//     PlcTask Inputs/GVL_iXlinker.EtherCAT_Master_EKxxxx.Beckhoff_EKM1xxx.Beckhoff_EKM1xxxEK1122.A_0004_EKM1101_0000_0019.MMS_Voltage_Us_In_Inputs.Status/Limit_2 <-> MMS Voltage Us In Inputs/Status/Limit 2
//     PlcTask Inputs/GVL_iXlinker.EtherCAT_Master_EKxxxx.Beckhoff_EKM1xxx.Beckhoff_EKM1xxxEK1122.A_0004_EKM1101_0000_0019.MMS_Voltage_Us_In_Inputs.Status/Error <-> MMS Voltage Us In Inputs/Status/Error
//     PlcTask Inputs/GVL_iXlinker.EtherCAT_Master_EKxxxx.Beckhoff_EKM1xxx.Beckhoff_EKM1xxxEK1122.A_0004_EKM1101_0000_0019.MMS_Voltage_Us_In_Inputs.Status/TxPDO_State <-> MMS Voltage Us In Inputs/Status/TxPDO State
//     PlcTask Inputs/GVL_iXlinker.EtherCAT_Master_EKxxxx.Beckhoff_EKM1xxx.Beckhoff_EKM1xxxEK1122.A_0004_EKM1101_0000_0019.MMS_Voltage_Us_In_Inputs.Status/TxPDO_Toggle <-> MMS Voltage Us In Inputs/Status/TxPDO Toggle
//     PlcTask Inputs/GVL_iXlinker.EtherCAT_Master_EKxxxx.Beckhoff_EKM1xxx.Beckhoff_EKM1xxxEK1122.A_0004_EKM1101_0000_0019.MMS_Voltage_Us_In_Inputs.Value <-> MMS Voltage Us In Inputs/Value
//     PlcTask Inputs/GVL_iXlinker.EtherCAT_Master_EKxxxx.Beckhoff_EKM1xxx.Beckhoff_EKM1xxxEK1122.A_0004_EKM1101_0000_0019.MMS_Voltage_Up_In_Inputs.Status/Underrange <-> MMS Voltage Up In Inputs/Status/Underrange
//     PlcTask Inputs/GVL_iXlinker.EtherCAT_Master_EKxxxx.Beckhoff_EKM1xxx.Beckhoff_EKM1xxxEK1122.A_0004_EKM1101_0000_0019.MMS_Voltage_Up_In_Inputs.Status/Overrange <-> MMS Voltage Up In Inputs/Status/Overrange
//     PlcTask Inputs/GVL_iXlinker.EtherCAT_Master_EKxxxx.Beckhoff_EKM1xxx.Beckhoff_EKM1xxxEK1122.A_0004_EKM1101_0000_0019.MMS_Voltage_Up_In_Inputs.Status/Limit_1 <-> MMS Voltage Up In Inputs/Status/Limit 1
//     PlcTask Inputs/GVL_iXlinker.EtherCAT_Master_EKxxxx.Beckhoff_EKM1xxx.Beckhoff_EKM1xxxEK1122.A_0004_EKM1101_0000_0019.MMS_Voltage_Up_In_Inputs.Status/Limit_2 <-> MMS Voltage Up In Inputs/Status/Limit 2
//     PlcTask Inputs/GVL_iXlinker.EtherCAT_Master_EKxxxx.Beckhoff_EKM1xxx.Beckhoff_EKM1xxxEK1122.A_0004_EKM1101_0000_0019.MMS_Voltage_Up_In_Inputs.Status/Error <-> MMS Voltage Up In Inputs/Status/Error
//     PlcTask Inputs/GVL_iXlinker.EtherCAT_Master_EKxxxx.Beckhoff_EKM1xxx.Beckhoff_EKM1xxxEK1122.A_0004_EKM1101_0000_0019.MMS_Voltage_Up_In_Inputs.Status/TxPDO_State <-> MMS Voltage Up In Inputs/Status/TxPDO State
//     PlcTask Inputs/GVL_iXlinker.EtherCAT_Master_EKxxxx.Beckhoff_EKM1xxx.Beckhoff_EKM1xxxEK1122.A_0004_EKM1101_0000_0019.MMS_Voltage_Up_In_Inputs.Status/TxPDO_Toggle <-> MMS Voltage Up In Inputs/Status/TxPDO Toggle
//     PlcTask Inputs/GVL_iXlinker.EtherCAT_Master_EKxxxx.Beckhoff_EKM1xxx.Beckhoff_EKM1xxxEK1122.A_0004_EKM1101_0000_0019.MMS_Voltage_Up_In_Inputs.Value <-> MMS Voltage Up In Inputs/Value
//     PlcTask Inputs/GVL_iXlinker.EtherCAT_Master_EKxxxx.Beckhoff_EKM1xxx.Beckhoff_EKM1xxxEK1122.A_0004_EKM1101_0000_0019.MMS_Voltage_Up_Out_Inputs.Status/Underrange <-> MMS Voltage Up Out Inputs/Status/Underrange
//     PlcTask Inputs/GVL_iXlinker.EtherCAT_Master_EKxxxx.Beckhoff_EKM1xxx.Beckhoff_EKM1xxxEK1122.A_0004_EKM1101_0000_0019.MMS_Voltage_Up_Out_Inputs.Status/Overrange <-> MMS Voltage Up Out Inputs/Status/Overrange
//     PlcTask Inputs/GVL_iXlinker.EtherCAT_Master_EKxxxx.Beckhoff_EKM1xxx.Beckhoff_EKM1xxxEK1122.A_0004_EKM1101_0000_0019.MMS_Voltage_Up_Out_Inputs.Status/Limit_1 <-> MMS Voltage Up Out Inputs/Status/Limit 1
//     PlcTask Inputs/GVL_iXlinker.EtherCAT_Master_EKxxxx.Beckhoff_EKM1xxx.Beckhoff_EKM1xxxEK1122.A_0004_EKM1101_0000_0019.MMS_Voltage_Up_Out_Inputs.Status/Limit_2 <-> MMS Voltage Up Out Inputs/Status/Limit 2
//     PlcTask Inputs/GVL_iXlinker.EtherCAT_Master_EKxxxx.Beckhoff_EKM1xxx.Beckhoff_EKM1xxxEK1122.A_0004_EKM1101_0000_0019.MMS_Voltage_Up_Out_Inputs.Status/Error <-> MMS Voltage Up Out Inputs/Status/Error
//     PlcTask Inputs/GVL_iXlinker.EtherCAT_Master_EKxxxx.Beckhoff_EKM1xxx.Beckhoff_EKM1xxxEK1122.A_0004_EKM1101_0000_0019.MMS_Voltage_Up_Out_Inputs.Status/TxPDO_State <-> MMS Voltage Up Out Inputs/Status/TxPDO State
//     PlcTask Inputs/GVL_iXlinker.EtherCAT_Master_EKxxxx.Beckhoff_EKM1xxx.Beckhoff_EKM1xxxEK1122.A_0004_EKM1101_0000_0019.MMS_Voltage_Up_Out_Inputs.Status/TxPDO_Toggle <-> MMS Voltage Up Out Inputs/Status/TxPDO Toggle
//     PlcTask Inputs/GVL_iXlinker.EtherCAT_Master_EKxxxx.Beckhoff_EKM1xxx.Beckhoff_EKM1xxxEK1122.A_0004_EKM1101_0000_0019.MMS_Voltage_Up_Out_Inputs.Value <-> MMS Voltage Up Out Inputs/Value
//     PlcTask Outputs/GVL_iXlinker.EtherCAT_Master_EKxxxx.Beckhoff_EKM1xxx.Beckhoff_EKM1xxxEK1122.A_0004_EKM1101_0000_0019.MMS_Device_Outputs.Control/Up_Out_OFF <-> MMS Device Outputs/Control/Up Out OFF
//     PlcTask Inputs/GVL_iXlinker.EtherCAT_Master_EKxxxx.Beckhoff_EKM1xxx.Beckhoff_EKM1xxxEK1122.A_0004_EKM1101_0000_0019.WcState.WcState <-> WcState/WcState
//     PlcTask Inputs/GVL_iXlinker.EtherCAT_Master_EKxxxx.Beckhoff_EKM1xxx.Beckhoff_EKM1xxxEK1122.A_0004_EKM1101_0000_0019.WcState.InputToggle <-> WcState/InputToggle
//     PlcTask Inputs/GVL_iXlinker.EtherCAT_Master_EKxxxx.Beckhoff_EKM1xxx.Beckhoff_EKM1xxxEK1122.A_0004_EKM1101_0000_0019.InfoData.AdsAddr <-> InfoData/AdsAddr
//     PlcTask Inputs/GVL_iXlinker.EtherCAT_Master_EKxxxx.Beckhoff_EKM1xxx.Beckhoff_EKM1xxxEK1122.A_0004_EKM1101_0000_0019.InfoData.DcOutputShift <-> InfoData/DcOutputShift
//     PlcTask Inputs/GVL_iXlinker.EtherCAT_Master_EKxxxx.Beckhoff_EKM1xxx.Beckhoff_EKM1xxxEK1122.A_0004_EKM1101_0000_0019.InfoData.DcInputShift <-> InfoData/DcInputShift
//     PlcTask Inputs/GVL_iXlinker.EtherCAT_Master_EKxxxx.Beckhoff_EKM1xxx.Beckhoff_EKM1xxxEK1122.A_0004_EKM1101_0000_0019.InfoData.State <-> InfoData/State
//   PLC/PLC Instance <-> EtherCAT Master EKxxxx/Beckhoff EKM1xxx/Beckhoff EKM1xxxEK1122/A_0005(EKM1101-0000-0020)
//     PlcTask Inputs/GVL_iXlinker.EtherCAT_Master_EKxxxx.Beckhoff_EKM1xxx.Beckhoff_EKM1xxxEK1122.A_0005_EKM1101_0000_0020.MMS_Device_Inputs.Status/Diag <-> MMS Device Inputs/Status/Diag
//     PlcTask Inputs/GVL_iXlinker.EtherCAT_Master_EKxxxx.Beckhoff_EKM1xxx.Beckhoff_EKM1xxxEK1122.A_0005_EKM1101_0000_0020.MMS_Device_Inputs.Status/Error <-> MMS Device Inputs/Status/Error
//     PlcTask Inputs/GVL_iXlinker.EtherCAT_Master_EKxxxx.Beckhoff_EKM1xxx.Beckhoff_EKM1xxxEK1122.A_0005_EKM1101_0000_0020.MMS_Device_Inputs.Status/Input_cycle_Counter <-> MMS Device Inputs/Status/Input cycle Counter
//     PlcTask Inputs/GVL_iXlinker.EtherCAT_Master_EKxxxx.Beckhoff_EKM1xxx.Beckhoff_EKM1xxxEK1122.A_0005_EKM1101_0000_0020.MMS_Device_Inputs.Status/TxPDO_State <-> MMS Device Inputs/Status/TxPDO State
//     PlcTask Inputs/GVL_iXlinker.EtherCAT_Master_EKxxxx.Beckhoff_EKM1xxx.Beckhoff_EKM1xxxEK1122.A_0005_EKM1101_0000_0020.MMS_Device_Inputs.Status/ID <-> MMS Device Inputs/Status/ID
//     PlcTask Inputs/GVL_iXlinker.EtherCAT_Master_EKxxxx.Beckhoff_EKM1xxx.Beckhoff_EKM1xxxEK1122.A_0005_EKM1101_0000_0020.MMS_Acceleration_Status.Status/Error <-> MMS Acceleration Status/Status/Error
//     PlcTask Inputs/GVL_iXlinker.EtherCAT_Master_EKxxxx.Beckhoff_EKM1xxx.Beckhoff_EKM1xxxEK1122.A_0005_EKM1101_0000_0020.MMS_Acceleration_Status.Status/Underrange <-> MMS Acceleration Status/Status/Underrange
//     PlcTask Inputs/GVL_iXlinker.EtherCAT_Master_EKxxxx.Beckhoff_EKM1xxx.Beckhoff_EKM1xxxEK1122.A_0005_EKM1101_0000_0020.MMS_Acceleration_Status.Status/Overrange <-> MMS Acceleration Status/Status/Overrange
//     PlcTask Inputs/GVL_iXlinker.EtherCAT_Master_EKxxxx.Beckhoff_EKM1xxx.Beckhoff_EKM1xxxEK1122.A_0005_EKM1101_0000_0020.MMS_Acceleration_Status.Status/Diag <-> MMS Acceleration Status/Status/Diag
//     PlcTask Inputs/GVL_iXlinker.EtherCAT_Master_EKxxxx.Beckhoff_EKM1xxx.Beckhoff_EKM1xxxEK1122.A_0005_EKM1101_0000_0020.MMS_Acceleration_Status.Status/Sensor_Ovr <-> MMS Acceleration Status/Status/Sensor Ovr
//     PlcTask Inputs/GVL_iXlinker.EtherCAT_Master_EKxxxx.Beckhoff_EKM1xxx.Beckhoff_EKM1xxxEK1122.A_0005_EKM1101_0000_0020.MMS_Acceleration_Status.Status/Overrun <-> MMS Acceleration Status/Status/Overrun
//     PlcTask Inputs/GVL_iXlinker.EtherCAT_Master_EKxxxx.Beckhoff_EKM1xxx.Beckhoff_EKM1xxxEK1122.A_0005_EKM1101_0000_0020.MMS_Acceleration_Status.Status/TxPDO_State <-> MMS Acceleration Status/Status/TxPDO State
//     PlcTask Inputs/GVL_iXlinker.EtherCAT_Master_EKxxxx.Beckhoff_EKM1xxx.Beckhoff_EKM1xxxEK1122.A_0005_EKM1101_0000_0020.MMS_Acceleration_Status.Number_of_samples <-> MMS Acceleration Status/Number of samples
//     PlcTask Inputs/GVL_iXlinker.EtherCAT_Master_EKxxxx.Beckhoff_EKM1xxx.Beckhoff_EKM1xxxEK1122.A_0005_EKM1101_0000_0020.MMS_Acceleration_X_Axis.Value <-> MMS Acceleration X-Axis/Value
//     PlcTask Inputs/GVL_iXlinker.EtherCAT_Master_EKxxxx.Beckhoff_EKM1xxx.Beckhoff_EKM1xxxEK1122.A_0005_EKM1101_0000_0020.MMS_Acceleration_Y_Axis.Value <-> MMS Acceleration Y-Axis/Value
//     PlcTask Inputs/GVL_iXlinker.EtherCAT_Master_EKxxxx.Beckhoff_EKM1xxx.Beckhoff_EKM1xxxEK1122.A_0005_EKM1101_0000_0020.MMS_Acceleration_Z_Axis.Value <-> MMS Acceleration Z-Axis/Value
//     PlcTask Inputs/GVL_iXlinker.EtherCAT_Master_EKxxxx.Beckhoff_EKM1xxx.Beckhoff_EKM1xxxEK1122.A_0005_EKM1101_0000_0020.MMS_Acceleration_Timestamp.Timestamp <-> MMS Acceleration Timestamp/Timestamp
//     PlcTask Inputs/GVL_iXlinker.EtherCAT_Master_EKxxxx.Beckhoff_EKM1xxx.Beckhoff_EKM1xxxEK1122.A_0005_EKM1101_0000_0020.MMS_Voltage_Us_In_Inputs.Status/Underrange <-> MMS Voltage Us In Inputs/Status/Underrange
//     PlcTask Inputs/GVL_iXlinker.EtherCAT_Master_EKxxxx.Beckhoff_EKM1xxx.Beckhoff_EKM1xxxEK1122.A_0005_EKM1101_0000_0020.MMS_Voltage_Us_In_Inputs.Status/Overrange <-> MMS Voltage Us In Inputs/Status/Overrange
//     PlcTask Inputs/GVL_iXlinker.EtherCAT_Master_EKxxxx.Beckhoff_EKM1xxx.Beckhoff_EKM1xxxEK1122.A_0005_EKM1101_0000_0020.MMS_Voltage_Us_In_Inputs.Status/Limit_1 <-> MMS Voltage Us In Inputs/Status/Limit 1
//     PlcTask Inputs/GVL_iXlinker.EtherCAT_Master_EKxxxx.Beckhoff_EKM1xxx.Beckhoff_EKM1xxxEK1122.A_0005_EKM1101_0000_0020.MMS_Voltage_Us_In_Inputs.Status/Limit_2 <-> MMS Voltage Us In Inputs/Status/Limit 2
//     PlcTask Inputs/GVL_iXlinker.EtherCAT_Master_EKxxxx.Beckhoff_EKM1xxx.Beckhoff_EKM1xxxEK1122.A_0005_EKM1101_0000_0020.MMS_Voltage_Us_In_Inputs.Status/Error <-> MMS Voltage Us In Inputs/Status/Error
//     PlcTask Inputs/GVL_iXlinker.EtherCAT_Master_EKxxxx.Beckhoff_EKM1xxx.Beckhoff_EKM1xxxEK1122.A_0005_EKM1101_0000_0020.MMS_Voltage_Us_In_Inputs.Status/TxPDO_State <-> MMS Voltage Us In Inputs/Status/TxPDO State
//     PlcTask Inputs/GVL_iXlinker.EtherCAT_Master_EKxxxx.Beckhoff_EKM1xxx.Beckhoff_EKM1xxxEK1122.A_0005_EKM1101_0000_0020.MMS_Voltage_Us_In_Inputs.Status/TxPDO_Toggle <-> MMS Voltage Us In Inputs/Status/TxPDO Toggle
//     PlcTask Inputs/GVL_iXlinker.EtherCAT_Master_EKxxxx.Beckhoff_EKM1xxx.Beckhoff_EKM1xxxEK1122.A_0005_EKM1101_0000_0020.MMS_Voltage_Us_In_Inputs.Value <-> MMS Voltage Us In Inputs/Value
//     PlcTask Inputs/GVL_iXlinker.EtherCAT_Master_EKxxxx.Beckhoff_EKM1xxx.Beckhoff_EKM1xxxEK1122.A_0005_EKM1101_0000_0020.MMS_Voltage_Up_In_Inputs.Status/Underrange <-> MMS Voltage Up In Inputs/Status/Underrange
//     PlcTask Inputs/GVL_iXlinker.EtherCAT_Master_EKxxxx.Beckhoff_EKM1xxx.Beckhoff_EKM1xxxEK1122.A_0005_EKM1101_0000_0020.MMS_Voltage_Up_In_Inputs.Status/Overrange <-> MMS Voltage Up In Inputs/Status/Overrange
//     PlcTask Inputs/GVL_iXlinker.EtherCAT_Master_EKxxxx.Beckhoff_EKM1xxx.Beckhoff_EKM1xxxEK1122.A_0005_EKM1101_0000_0020.MMS_Voltage_Up_In_Inputs.Status/Limit_1 <-> MMS Voltage Up In Inputs/Status/Limit 1
//     PlcTask Inputs/GVL_iXlinker.EtherCAT_Master_EKxxxx.Beckhoff_EKM1xxx.Beckhoff_EKM1xxxEK1122.A_0005_EKM1101_0000_0020.MMS_Voltage_Up_In_Inputs.Status/Limit_2 <-> MMS Voltage Up In Inputs/Status/Limit 2
//     PlcTask Inputs/GVL_iXlinker.EtherCAT_Master_EKxxxx.Beckhoff_EKM1xxx.Beckhoff_EKM1xxxEK1122.A_0005_EKM1101_0000_0020.MMS_Voltage_Up_In_Inputs.Status/Error <-> MMS Voltage Up In Inputs/Status/Error
//     PlcTask Inputs/GVL_iXlinker.EtherCAT_Master_EKxxxx.Beckhoff_EKM1xxx.Beckhoff_EKM1xxxEK1122.A_0005_EKM1101_0000_0020.MMS_Voltage_Up_In_Inputs.Status/TxPDO_State <-> MMS Voltage Up In Inputs/Status/TxPDO State
//     PlcTask Inputs/GVL_iXlinker.EtherCAT_Master_EKxxxx.Beckhoff_EKM1xxx.Beckhoff_EKM1xxxEK1122.A_0005_EKM1101_0000_0020.MMS_Voltage_Up_In_Inputs.Status/TxPDO_Toggle <-> MMS Voltage Up In Inputs/Status/TxPDO Toggle
//     PlcTask Inputs/GVL_iXlinker.EtherCAT_Master_EKxxxx.Beckhoff_EKM1xxx.Beckhoff_EKM1xxxEK1122.A_0005_EKM1101_0000_0020.MMS_Voltage_Up_In_Inputs.Value <-> MMS Voltage Up In Inputs/Value
//     PlcTask Inputs/GVL_iXlinker.EtherCAT_Master_EKxxxx.Beckhoff_EKM1xxx.Beckhoff_EKM1xxxEK1122.A_0005_EKM1101_0000_0020.MMS_Voltage_Up_Out_Inputs.Status/Underrange <-> MMS Voltage Up Out Inputs/Status/Underrange
//     PlcTask Inputs/GVL_iXlinker.EtherCAT_Master_EKxxxx.Beckhoff_EKM1xxx.Beckhoff_EKM1xxxEK1122.A_0005_EKM1101_0000_0020.MMS_Voltage_Up_Out_Inputs.Status/Overrange <-> MMS Voltage Up Out Inputs/Status/Overrange
//     PlcTask Inputs/GVL_iXlinker.EtherCAT_Master_EKxxxx.Beckhoff_EKM1xxx.Beckhoff_EKM1xxxEK1122.A_0005_EKM1101_0000_0020.MMS_Voltage_Up_Out_Inputs.Status/Limit_1 <-> MMS Voltage Up Out Inputs/Status/Limit 1
//     PlcTask Inputs/GVL_iXlinker.EtherCAT_Master_EKxxxx.Beckhoff_EKM1xxx.Beckhoff_EKM1xxxEK1122.A_0005_EKM1101_0000_0020.MMS_Voltage_Up_Out_Inputs.Status/Limit_2 <-> MMS Voltage Up Out Inputs/Status/Limit 2
//     PlcTask Inputs/GVL_iXlinker.EtherCAT_Master_EKxxxx.Beckhoff_EKM1xxx.Beckhoff_EKM1xxxEK1122.A_0005_EKM1101_0000_0020.MMS_Voltage_Up_Out_Inputs.Status/Error <-> MMS Voltage Up Out Inputs/Status/Error
//     PlcTask Inputs/GVL_iXlinker.EtherCAT_Master_EKxxxx.Beckhoff_EKM1xxx.Beckhoff_EKM1xxxEK1122.A_0005_EKM1101_0000_0020.MMS_Voltage_Up_Out_Inputs.Status/TxPDO_State <-> MMS Voltage Up Out Inputs/Status/TxPDO State
//     PlcTask Inputs/GVL_iXlinker.EtherCAT_Master_EKxxxx.Beckhoff_EKM1xxx.Beckhoff_EKM1xxxEK1122.A_0005_EKM1101_0000_0020.MMS_Voltage_Up_Out_Inputs.Status/TxPDO_Toggle <-> MMS Voltage Up Out Inputs/Status/TxPDO Toggle
//     PlcTask Inputs/GVL_iXlinker.EtherCAT_Master_EKxxxx.Beckhoff_EKM1xxx.Beckhoff_EKM1xxxEK1122.A_0005_EKM1101_0000_0020.MMS_Voltage_Up_Out_Inputs.Value <-> MMS Voltage Up Out Inputs/Value
//     PlcTask Outputs/GVL_iXlinker.EtherCAT_Master_EKxxxx.Beckhoff_EKM1xxx.Beckhoff_EKM1xxxEK1122.A_0005_EKM1101_0000_0020.MMS_Device_Outputs.Control/Up_Out_OFF <-> MMS Device Outputs/Control/Up Out OFF
//     PlcTask Inputs/GVL_iXlinker.EtherCAT_Master_EKxxxx.Beckhoff_EKM1xxx.Beckhoff_EKM1xxxEK1122.A_0005_EKM1101_0000_0020.WcState.WcState <-> WcState/WcState
//     PlcTask Inputs/GVL_iXlinker.EtherCAT_Master_EKxxxx.Beckhoff_EKM1xxx.Beckhoff_EKM1xxxEK1122.A_0005_EKM1101_0000_0020.WcState.InputToggle <-> WcState/InputToggle
//     PlcTask Inputs/GVL_iXlinker.EtherCAT_Master_EKxxxx.Beckhoff_EKM1xxx.Beckhoff_EKM1xxxEK1122.A_0005_EKM1101_0000_0020.InfoData.AdsAddr <-> InfoData/AdsAddr
//     PlcTask Inputs/GVL_iXlinker.EtherCAT_Master_EKxxxx.Beckhoff_EKM1xxx.Beckhoff_EKM1xxxEK1122.A_0005_EKM1101_0000_0020.InfoData.DcOutputShift <-> InfoData/DcOutputShift
//     PlcTask Inputs/GVL_iXlinker.EtherCAT_Master_EKxxxx.Beckhoff_EKM1xxx.Beckhoff_EKM1xxxEK1122.A_0005_EKM1101_0000_0020.InfoData.DcInputShift <-> InfoData/DcInputShift
//     PlcTask Inputs/GVL_iXlinker.EtherCAT_Master_EKxxxx.Beckhoff_EKM1xxx.Beckhoff_EKM1xxxEK1122.A_0005_EKM1101_0000_0020.InfoData.State <-> InfoData/State
//   PLC/PLC Instance <-> EtherCAT Master EKxxxx/Beckhoff EKx9xx
//     PlcTask Inputs/GVL_iXlinker.EtherCAT_Master_EKxxxx.Beckhoff_EKx9xx.InfoData.State <-> InfoData/State
//   PLC/PLC Instance <-> EtherCAT Master EKxxxx/Beckhoff EKx9xx/Beckhoff EKx9xxEK1122
//     PlcTask Inputs/GVL_iXlinker.EtherCAT_Master_EKxxxx.Beckhoff_EKx9xx.Beckhoff_EKx9xxEK1122.InfoData.State <-> InfoData/State
//   PLC/PLC Instance <-> EtherCAT Master EKxxxx/Beckhoff EKx9xx/Beckhoff EKx9xxEK1122/Beckhoff EKx9xxsub EK1100
//     PlcTask Inputs/GVL_iXlinker.EtherCAT_Master_EKxxxx.Beckhoff_EKx9xx.Beckhoff_EKx9xxEK1122.Beckhoff_EKx9xxsub_EK1100.InfoData.State <-> InfoData/State
//   PLC/PLC Instance <-> EtherCAT Master EKxxxx/Beckhoff EKx9xx/Beckhoff EKx9xxEK1122/A_0001(EK1960-0000-0019)
//     PlcTask Inputs/GVL_iXlinker.EtherCAT_Master_EKxxxx.Beckhoff_EKx9xx.Beckhoff_EKx9xxEK1122.A_0001_EK1960_0000_0019.Module_1_FSoE.FSoE_Inputs.FSOE/FSoE_Command <-> Module 1 (FSoE)/FSoE Inputs/FSOE/FSoE Command
//     PlcTask Inputs/GVL_iXlinker.EtherCAT_Master_EKxxxx.Beckhoff_EKx9xx.Beckhoff_EKx9xxEK1122.A_0001_EK1960_0000_0019.Module_1_FSoE.FSoE_Inputs.FSOE/FSOUT_Module_1_Module_Fault <-> Module 1 (FSoE)/FSoE Inputs/FSOE/FSOUT Module 1.Module Fault
//     PlcTask Inputs/GVL_iXlinker.EtherCAT_Master_EKxxxx.Beckhoff_EKx9xx.Beckhoff_EKx9xxEK1122.A_0001_EK1960_0000_0019.Module_1_FSoE.FSoE_Inputs.FSOE/FSOUT_Module_2_Module_Fault <-> Module 1 (FSoE)/FSoE Inputs/FSOE/FSOUT Module 2.Module Fault
//     PlcTask Inputs/GVL_iXlinker.EtherCAT_Master_EKxxxx.Beckhoff_EKx9xx.Beckhoff_EKx9xxEK1122.A_0001_EK1960_0000_0019.Module_1_FSoE.FSoE_Inputs.FSOE/FSOUT_Module_3_Module_Fault <-> Module 1 (FSoE)/FSoE Inputs/FSOE/FSOUT Module 3.Module Fault
//     PlcTask Inputs/GVL_iXlinker.EtherCAT_Master_EKxxxx.Beckhoff_EKx9xx.Beckhoff_EKx9xxEK1122.A_0001_EK1960_0000_0019.Module_1_FSoE.FSoE_Inputs.FSOE/FSOUT_Module_4_Module_Fault <-> Module 1 (FSoE)/FSoE Inputs/FSOE/FSOUT Module 4.Module Fault
//     PlcTask Inputs/GVL_iXlinker.EtherCAT_Master_EKxxxx.Beckhoff_EKx9xx.Beckhoff_EKx9xxEK1122.A_0001_EK1960_0000_0019.Module_1_FSoE.FSoE_Inputs.FSOE/FSOUT_Module_5_Module_Fault <-> Module 1 (FSoE)/FSoE Inputs/FSOE/FSOUT Module 5.Module Fault
//     PlcTask Inputs/GVL_iXlinker.EtherCAT_Master_EKxxxx.Beckhoff_EKx9xx.Beckhoff_EKx9xxEK1122.A_0001_EK1960_0000_0019.Module_1_FSoE.FSoE_Inputs.FSOE/FSOUT_Module_6_Module_Fault <-> Module 1 (FSoE)/FSoE Inputs/FSOE/FSOUT Module 6.Module Fault
//     PlcTask Inputs/GVL_iXlinker.EtherCAT_Master_EKxxxx.Beckhoff_EKx9xx.Beckhoff_EKx9xxEK1122.A_0001_EK1960_0000_0019.Module_1_FSoE.FSoE_Inputs.FSOE/FSIN_Module_1_Channel_1_Input <-> Module 1 (FSoE)/FSoE Inputs/FSOE/FSIN Module 1.Channel 1.Input
//     PlcTask Inputs/GVL_iXlinker.EtherCAT_Master_EKxxxx.Beckhoff_EKx9xx.Beckhoff_EKx9xxEK1122.A_0001_EK1960_0000_0019.Module_1_FSoE.FSoE_Inputs.FSOE/FSIN_Module_1_Channel_2_Input <-> Module 1 (FSoE)/FSoE Inputs/FSOE/FSIN Module 1.Channel 2.Input
//     PlcTask Inputs/GVL_iXlinker.EtherCAT_Master_EKxxxx.Beckhoff_EKx9xx.Beckhoff_EKx9xxEK1122.A_0001_EK1960_0000_0019.Module_1_FSoE.FSoE_Inputs.FSOE/FSIN_Module_2_Channel_1_Input <-> Module 1 (FSoE)/FSoE Inputs/FSOE/FSIN Module 2.Channel 1.Input
//     PlcTask Inputs/GVL_iXlinker.EtherCAT_Master_EKxxxx.Beckhoff_EKx9xx.Beckhoff_EKx9xxEK1122.A_0001_EK1960_0000_0019.Module_1_FSoE.FSoE_Inputs.FSOE/FSIN_Module_2_Channel_2_Input <-> Module 1 (FSoE)/FSoE Inputs/FSOE/FSIN Module 2.Channel 2.Input
//     PlcTask Inputs/GVL_iXlinker.EtherCAT_Master_EKxxxx.Beckhoff_EKx9xx.Beckhoff_EKx9xxEK1122.A_0001_EK1960_0000_0019.Module_1_FSoE.FSoE_Inputs.FSOE/FSIN_Module_3_Channel_1_Input <-> Module 1 (FSoE)/FSoE Inputs/FSOE/FSIN Module 3.Channel 1.Input
//     PlcTask Inputs/GVL_iXlinker.EtherCAT_Master_EKxxxx.Beckhoff_EKx9xx.Beckhoff_EKx9xxEK1122.A_0001_EK1960_0000_0019.Module_1_FSoE.FSoE_Inputs.FSOE/FSIN_Module_3_Channel_2_Input <-> Module 1 (FSoE)/FSoE Inputs/FSOE/FSIN Module 3.Channel 2.Input
//     PlcTask Inputs/GVL_iXlinker.EtherCAT_Master_EKxxxx.Beckhoff_EKx9xx.Beckhoff_EKx9xxEK1122.A_0001_EK1960_0000_0019.Module_1_FSoE.FSoE_Inputs.FSOE/FSIN_Module_4_Channel_1_Input <-> Module 1 (FSoE)/FSoE Inputs/FSOE/FSIN Module 4.Channel 1.Input
//     PlcTask Inputs/GVL_iXlinker.EtherCAT_Master_EKxxxx.Beckhoff_EKx9xx.Beckhoff_EKx9xxEK1122.A_0001_EK1960_0000_0019.Module_1_FSoE.FSoE_Inputs.FSOE/FSIN_Module_4_Channel_2_Input <-> Module 1 (FSoE)/FSoE Inputs/FSOE/FSIN Module 4.Channel 2.Input
//     PlcTask Inputs/GVL_iXlinker.EtherCAT_Master_EKxxxx.Beckhoff_EKx9xx.Beckhoff_EKx9xxEK1122.A_0001_EK1960_0000_0019.Module_1_FSoE.FSoE_Inputs.FSOE/FSIN_Module_5_Channel_1_Input <-> Module 1 (FSoE)/FSoE Inputs/FSOE/FSIN Module 5.Channel 1.Input
//     PlcTask Inputs/GVL_iXlinker.EtherCAT_Master_EKxxxx.Beckhoff_EKx9xx.Beckhoff_EKx9xxEK1122.A_0001_EK1960_0000_0019.Module_1_FSoE.FSoE_Inputs.FSOE/FSIN_Module_5_Channel_2_Input <-> Module 1 (FSoE)/FSoE Inputs/FSOE/FSIN Module 5.Channel 2.Input
//     PlcTask Inputs/GVL_iXlinker.EtherCAT_Master_EKxxxx.Beckhoff_EKx9xx.Beckhoff_EKx9xxEK1122.A_0001_EK1960_0000_0019.Module_1_FSoE.FSoE_Inputs.FSOE/FSIN_Module_6_Channel_1_Input <-> Module 1 (FSoE)/FSoE Inputs/FSOE/FSIN Module 6.Channel 1.Input
//     PlcTask Inputs/GVL_iXlinker.EtherCAT_Master_EKxxxx.Beckhoff_EKx9xx.Beckhoff_EKx9xxEK1122.A_0001_EK1960_0000_0019.Module_1_FSoE.FSoE_Inputs.FSOE/FSIN_Module_6_Channel_2_Input <-> Module 1 (FSoE)/FSoE Inputs/FSOE/FSIN Module 6.Channel 2.Input
//     PlcTask Inputs/GVL_iXlinker.EtherCAT_Master_EKxxxx.Beckhoff_EKx9xx.Beckhoff_EKx9xxEK1122.A_0001_EK1960_0000_0019.Module_1_FSoE.FSoE_Inputs.FSOE/FSIN_Module_7_Channel_1_Input <-> Module 1 (FSoE)/FSoE Inputs/FSOE/FSIN Module 7.Channel 1.Input
//     PlcTask Inputs/GVL_iXlinker.EtherCAT_Master_EKxxxx.Beckhoff_EKx9xx.Beckhoff_EKx9xxEK1122.A_0001_EK1960_0000_0019.Module_1_FSoE.FSoE_Inputs.FSOE/FSIN_Module_7_Channel_2_Input <-> Module 1 (FSoE)/FSoE Inputs/FSOE/FSIN Module 7.Channel 2.Input
//     PlcTask Inputs/GVL_iXlinker.EtherCAT_Master_EKxxxx.Beckhoff_EKx9xx.Beckhoff_EKx9xxEK1122.A_0001_EK1960_0000_0019.Module_1_FSoE.FSoE_Inputs.FSOE/FSIN_Module_8_Channel_1_Input <-> Module 1 (FSoE)/FSoE Inputs/FSOE/FSIN Module 8.Channel 1.Input
//     PlcTask Inputs/GVL_iXlinker.EtherCAT_Master_EKxxxx.Beckhoff_EKx9xx.Beckhoff_EKx9xxEK1122.A_0001_EK1960_0000_0019.Module_1_FSoE.FSoE_Inputs.FSOE/FSIN_Module_8_Channel_2_Input <-> Module 1 (FSoE)/FSoE Inputs/FSOE/FSIN Module 8.Channel 2.Input
//     PlcTask Inputs/GVL_iXlinker.EtherCAT_Master_EKxxxx.Beckhoff_EKx9xx.Beckhoff_EKx9xxEK1122.A_0001_EK1960_0000_0019.Module_1_FSoE.FSoE_Inputs.FSOE/FSIN_Module_9_Channel_1_Input <-> Module 1 (FSoE)/FSoE Inputs/FSOE/FSIN Module 9.Channel 1.Input
//     PlcTask Inputs/GVL_iXlinker.EtherCAT_Master_EKxxxx.Beckhoff_EKx9xx.Beckhoff_EKx9xxEK1122.A_0001_EK1960_0000_0019.Module_1_FSoE.FSoE_Inputs.FSOE/FSIN_Module_9_Channel_2_Input <-> Module 1 (FSoE)/FSoE Inputs/FSOE/FSIN Module 9.Channel 2.Input
//     PlcTask Inputs/GVL_iXlinker.EtherCAT_Master_EKxxxx.Beckhoff_EKx9xx.Beckhoff_EKx9xxEK1122.A_0001_EK1960_0000_0019.Module_1_FSoE.FSoE_Inputs.FSOE/FSIN_Module_10_Channel_1_Input <-> Module 1 (FSoE)/FSoE Inputs/FSOE/FSIN Module 10.Channel 1.Input
//     PlcTask Inputs/GVL_iXlinker.EtherCAT_Master_EKxxxx.Beckhoff_EKx9xx.Beckhoff_EKx9xxEK1122.A_0001_EK1960_0000_0019.Module_1_FSoE.FSoE_Inputs.FSOE/FSIN_Module_10_Channel_2_Input <-> Module 1 (FSoE)/FSoE Inputs/FSOE/FSIN Module 10.Channel 2.Input
//     PlcTask Inputs/GVL_iXlinker.EtherCAT_Master_EKxxxx.Beckhoff_EKx9xx.Beckhoff_EKx9xxEK1122.A_0001_EK1960_0000_0019.Module_1_FSoE.FSoE_Inputs.FSOE/FSIN_Module_1_Module_Fault <-> Module 1 (FSoE)/FSoE Inputs/FSOE/FSIN Module 1.Module Fault
//     PlcTask Inputs/GVL_iXlinker.EtherCAT_Master_EKxxxx.Beckhoff_EKx9xx.Beckhoff_EKx9xxEK1122.A_0001_EK1960_0000_0019.Module_1_FSoE.FSoE_Inputs.FSOE/FSIN_Module_2_Module_Fault <-> Module 1 (FSoE)/FSoE Inputs/FSOE/FSIN Module 2.Module Fault
//     PlcTask Inputs/GVL_iXlinker.EtherCAT_Master_EKxxxx.Beckhoff_EKx9xx.Beckhoff_EKx9xxEK1122.A_0001_EK1960_0000_0019.Module_1_FSoE.FSoE_Inputs.FSOE/FSIN_Module_3_Module_Fault <-> Module 1 (FSoE)/FSoE Inputs/FSOE/FSIN Module 3.Module Fault
//     PlcTask Inputs/GVL_iXlinker.EtherCAT_Master_EKxxxx.Beckhoff_EKx9xx.Beckhoff_EKx9xxEK1122.A_0001_EK1960_0000_0019.Module_1_FSoE.FSoE_Inputs.FSOE/FSIN_Module_4_Module_Fault <-> Module 1 (FSoE)/FSoE Inputs/FSOE/FSIN Module 4.Module Fault
//     PlcTask Inputs/GVL_iXlinker.EtherCAT_Master_EKxxxx.Beckhoff_EKx9xx.Beckhoff_EKx9xxEK1122.A_0001_EK1960_0000_0019.Module_1_FSoE.FSoE_Inputs.FSOE/FSIN_Module_5_Module_Fault <-> Module 1 (FSoE)/FSoE Inputs/FSOE/FSIN Module 5.Module Fault
//     PlcTask Inputs/GVL_iXlinker.EtherCAT_Master_EKxxxx.Beckhoff_EKx9xx.Beckhoff_EKx9xxEK1122.A_0001_EK1960_0000_0019.Module_1_FSoE.FSoE_Inputs.FSOE/FSIN_Module_6_Module_Fault <-> Module 1 (FSoE)/FSoE Inputs/FSOE/FSIN Module 6.Module Fault
//     PlcTask Inputs/GVL_iXlinker.EtherCAT_Master_EKxxxx.Beckhoff_EKx9xx.Beckhoff_EKx9xxEK1122.A_0001_EK1960_0000_0019.Module_1_FSoE.FSoE_Inputs.FSOE/FSIN_Module_7_Module_Fault <-> Module 1 (FSoE)/FSoE Inputs/FSOE/FSIN Module 7.Module Fault
//     PlcTask Inputs/GVL_iXlinker.EtherCAT_Master_EKxxxx.Beckhoff_EKx9xx.Beckhoff_EKx9xxEK1122.A_0001_EK1960_0000_0019.Module_1_FSoE.FSoE_Inputs.FSOE/FSIN_Module_8_Module_Fault <-> Module 1 (FSoE)/FSoE Inputs/FSOE/FSIN Module 8.Module Fault
//     PlcTask Inputs/GVL_iXlinker.EtherCAT_Master_EKxxxx.Beckhoff_EKx9xx.Beckhoff_EKx9xxEK1122.A_0001_EK1960_0000_0019.Module_1_FSoE.FSoE_Inputs.FSOE/FSoE_CRC_000 <-> Module 1 (FSoE)/FSoE Inputs/FSOE/FSoE CRC 000
//     PlcTask Inputs/GVL_iXlinker.EtherCAT_Master_EKxxxx.Beckhoff_EKx9xx.Beckhoff_EKx9xxEK1122.A_0001_EK1960_0000_0019.Module_1_FSoE.FSoE_Inputs.FSOE/FSoE_CRC_001 <-> Module 1 (FSoE)/FSoE Inputs/FSOE/FSoE CRC 001
//     PlcTask Inputs/GVL_iXlinker.EtherCAT_Master_EKxxxx.Beckhoff_EKx9xx.Beckhoff_EKx9xxEK1122.A_0001_EK1960_0000_0019.Module_1_FSoE.FSoE_Inputs.FSOE/FSoE_CRC_002 <-> Module 1 (FSoE)/FSoE Inputs/FSOE/FSoE CRC 002
//     PlcTask Inputs/GVL_iXlinker.EtherCAT_Master_EKxxxx.Beckhoff_EKx9xx.Beckhoff_EKx9xxEK1122.A_0001_EK1960_0000_0019.Module_1_FSoE.FSoE_Inputs.FSOE/FSIN_Module_9_Module_Fault_1 <-> Module 1 (FSoE)/FSoE Inputs/FSOE/FSIN Module 9.Module Fault 1
//     PlcTask Inputs/GVL_iXlinker.EtherCAT_Master_EKxxxx.Beckhoff_EKx9xx.Beckhoff_EKx9xxEK1122.A_0001_EK1960_0000_0019.Module_1_FSoE.FSoE_Inputs.FSOE/FSIN_Module_9_Module_Fault_2 <-> Module 1 (FSoE)/FSoE Inputs/FSOE/FSIN Module 9.Module Fault 2
//     PlcTask Inputs/GVL_iXlinker.EtherCAT_Master_EKxxxx.Beckhoff_EKx9xx.Beckhoff_EKx9xxEK1122.A_0001_EK1960_0000_0019.Module_1_FSoE.FSoE_Inputs.FSOE/FSIN_Module_10_Module_Fault_1 <-> Module 1 (FSoE)/FSoE Inputs/FSOE/FSIN Module 10.Module Fault 1
//     PlcTask Inputs/GVL_iXlinker.EtherCAT_Master_EKxxxx.Beckhoff_EKx9xx.Beckhoff_EKx9xxEK1122.A_0001_EK1960_0000_0019.Module_1_FSoE.FSoE_Inputs.FSOE/FSIN_Module_10_Module_Fault_2 <-> Module 1 (FSoE)/FSoE Inputs/FSOE/FSIN Module 10.Module Fault 2
//     PlcTask Inputs/GVL_iXlinker.EtherCAT_Master_EKxxxx.Beckhoff_EKx9xx.Beckhoff_EKx9xxEK1122.A_0001_EK1960_0000_0019.Module_1_FSoE.FSoE_Inputs.FSOE/FSoE_Connection_ID <-> Module 1 (FSoE)/FSoE Inputs/FSOE/FSoE Connection ID
//     PlcTask Outputs/GVL_iXlinker.EtherCAT_Master_EKxxxx.Beckhoff_EKx9xx.Beckhoff_EKx9xxEK1122.A_0001_EK1960_0000_0019.Module_1_FSoE.FSoE_Outputs.FSOE/FSoE_Command <-> Module 1 (FSoE)/FSoE Outputs/FSOE/FSoE Command
//     PlcTask Outputs/GVL_iXlinker.EtherCAT_Master_EKxxxx.Beckhoff_EKx9xx.Beckhoff_EKx9xxEK1122.A_0001_EK1960_0000_0019.Module_1_FSoE.FSoE_Outputs.FSOE/FSOUT_Module_1_Channel_1_Output <-> Module 1 (FSoE)/FSoE Outputs/FSOE/FSOUT Module 1.Channel 1.Output
//     PlcTask Outputs/GVL_iXlinker.EtherCAT_Master_EKxxxx.Beckhoff_EKx9xx.Beckhoff_EKx9xxEK1122.A_0001_EK1960_0000_0019.Module_1_FSoE.FSoE_Outputs.FSOE/FSOUT_Module_1_Channel_2_Output <-> Module 1 (FSoE)/FSoE Outputs/FSOE/FSOUT Module 1.Channel 2.Output
//     PlcTask Outputs/GVL_iXlinker.EtherCAT_Master_EKxxxx.Beckhoff_EKx9xx.Beckhoff_EKx9xxEK1122.A_0001_EK1960_0000_0019.Module_1_FSoE.FSoE_Outputs.FSOE/FSOUT_Module_1_Channel_3_Output <-> Module 1 (FSoE)/FSoE Outputs/FSOE/FSOUT Module 1.Channel 3.Output
//     PlcTask Outputs/GVL_iXlinker.EtherCAT_Master_EKxxxx.Beckhoff_EKx9xx.Beckhoff_EKx9xxEK1122.A_0001_EK1960_0000_0019.Module_1_FSoE.FSoE_Outputs.FSOE/FSOUT_Module_1_Channel_4_Output <-> Module 1 (FSoE)/FSoE Outputs/FSOE/FSOUT Module 1.Channel 4.Output
//     PlcTask Outputs/GVL_iXlinker.EtherCAT_Master_EKxxxx.Beckhoff_EKx9xx.Beckhoff_EKx9xxEK1122.A_0001_EK1960_0000_0019.Module_1_FSoE.FSoE_Outputs.FSOE/FSOUT_Module_2_Channel_1_Output <-> Module 1 (FSoE)/FSoE Outputs/FSOE/FSOUT Module 2.Channel 1.Output
//     PlcTask Outputs/GVL_iXlinker.EtherCAT_Master_EKxxxx.Beckhoff_EKx9xx.Beckhoff_EKx9xxEK1122.A_0001_EK1960_0000_0019.Module_1_FSoE.FSoE_Outputs.FSOE/FSOUT_Module_2_Channel_2_Output <-> Module 1 (FSoE)/FSoE Outputs/FSOE/FSOUT Module 2.Channel 2.Output
//     PlcTask Outputs/GVL_iXlinker.EtherCAT_Master_EKxxxx.Beckhoff_EKx9xx.Beckhoff_EKx9xxEK1122.A_0001_EK1960_0000_0019.Module_1_FSoE.FSoE_Outputs.FSOE/FSOUT_Module_2_Channel_3_Output <-> Module 1 (FSoE)/FSoE Outputs/FSOE/FSOUT Module 2.Channel 3.Output
//     PlcTask Outputs/GVL_iXlinker.EtherCAT_Master_EKxxxx.Beckhoff_EKx9xx.Beckhoff_EKx9xxEK1122.A_0001_EK1960_0000_0019.Module_1_FSoE.FSoE_Outputs.FSOE/FSOUT_Module_2_Channel_4_Output <-> Module 1 (FSoE)/FSoE Outputs/FSOE/FSOUT Module 2.Channel 4.Output
//     PlcTask Outputs/GVL_iXlinker.EtherCAT_Master_EKxxxx.Beckhoff_EKx9xx.Beckhoff_EKx9xxEK1122.A_0001_EK1960_0000_0019.Module_1_FSoE.FSoE_Outputs.FSOE/FSOUT_Module_3_Channel_1_Output <-> Module 1 (FSoE)/FSoE Outputs/FSOE/FSOUT Module 3.Channel 1.Output
//     PlcTask Outputs/GVL_iXlinker.EtherCAT_Master_EKxxxx.Beckhoff_EKx9xx.Beckhoff_EKx9xxEK1122.A_0001_EK1960_0000_0019.Module_1_FSoE.FSoE_Outputs.FSOE/FSOUT_Module_3_Channel_2_Output <-> Module 1 (FSoE)/FSoE Outputs/FSOE/FSOUT Module 3.Channel 2.Output
//     PlcTask Outputs/GVL_iXlinker.EtherCAT_Master_EKxxxx.Beckhoff_EKx9xx.Beckhoff_EKx9xxEK1122.A_0001_EK1960_0000_0019.Module_1_FSoE.FSoE_Outputs.FSOE/FSOUT_Module_3_Channel_3_Output <-> Module 1 (FSoE)/FSoE Outputs/FSOE/FSOUT Module 3.Channel 3.Output
//     PlcTask Outputs/GVL_iXlinker.EtherCAT_Master_EKxxxx.Beckhoff_EKx9xx.Beckhoff_EKx9xxEK1122.A_0001_EK1960_0000_0019.Module_1_FSoE.FSoE_Outputs.FSOE/FSOUT_Module_3_Channel_4_Output <-> Module 1 (FSoE)/FSoE Outputs/FSOE/FSOUT Module 3.Channel 4.Output
//     PlcTask Outputs/GVL_iXlinker.EtherCAT_Master_EKxxxx.Beckhoff_EKx9xx.Beckhoff_EKx9xxEK1122.A_0001_EK1960_0000_0019.Module_1_FSoE.FSoE_Outputs.FSOE/FSOUT_Module_4_Channel_1_Output <-> Module 1 (FSoE)/FSoE Outputs/FSOE/FSOUT Module 4.Channel 1.Output
//     PlcTask Outputs/GVL_iXlinker.EtherCAT_Master_EKxxxx.Beckhoff_EKx9xx.Beckhoff_EKx9xxEK1122.A_0001_EK1960_0000_0019.Module_1_FSoE.FSoE_Outputs.FSOE/FSOUT_Module_4_Channel_2_Output <-> Module 1 (FSoE)/FSoE Outputs/FSOE/FSOUT Module 4.Channel 2.Output
//     PlcTask Outputs/GVL_iXlinker.EtherCAT_Master_EKxxxx.Beckhoff_EKx9xx.Beckhoff_EKx9xxEK1122.A_0001_EK1960_0000_0019.Module_1_FSoE.FSoE_Outputs.FSOE/FSOUT_Module_4_Channel_3_Output <-> Module 1 (FSoE)/FSoE Outputs/FSOE/FSOUT Module 4.Channel 3.Output
//     PlcTask Outputs/GVL_iXlinker.EtherCAT_Master_EKxxxx.Beckhoff_EKx9xx.Beckhoff_EKx9xxEK1122.A_0001_EK1960_0000_0019.Module_1_FSoE.FSoE_Outputs.FSOE/FSOUT_Module_4_Channel_4_Output <-> Module 1 (FSoE)/FSoE Outputs/FSOE/FSOUT Module 4.Channel 4.Output
//     PlcTask Outputs/GVL_iXlinker.EtherCAT_Master_EKxxxx.Beckhoff_EKx9xx.Beckhoff_EKx9xxEK1122.A_0001_EK1960_0000_0019.Module_1_FSoE.FSoE_Outputs.FSOE/FSOUT_Module_5_Channel_1_Output <-> Module 1 (FSoE)/FSoE Outputs/FSOE/FSOUT Module 5.Channel 1.Output
//     PlcTask Outputs/GVL_iXlinker.EtherCAT_Master_EKxxxx.Beckhoff_EKx9xx.Beckhoff_EKx9xxEK1122.A_0001_EK1960_0000_0019.Module_1_FSoE.FSoE_Outputs.FSOE/FSOUT_Module_5_Channel_2_Output <-> Module 1 (FSoE)/FSoE Outputs/FSOE/FSOUT Module 5.Channel 2.Output
//     PlcTask Outputs/GVL_iXlinker.EtherCAT_Master_EKxxxx.Beckhoff_EKx9xx.Beckhoff_EKx9xxEK1122.A_0001_EK1960_0000_0019.Module_1_FSoE.FSoE_Outputs.FSOE/FSOUT_Module_5_Channel_3_Output <-> Module 1 (FSoE)/FSoE Outputs/FSOE/FSOUT Module 5.Channel 3.Output
//     PlcTask Outputs/GVL_iXlinker.EtherCAT_Master_EKxxxx.Beckhoff_EKx9xx.Beckhoff_EKx9xxEK1122.A_0001_EK1960_0000_0019.Module_1_FSoE.FSoE_Outputs.FSOE/FSOUT_Module_5_Channel_4_Output <-> Module 1 (FSoE)/FSoE Outputs/FSOE/FSOUT Module 5.Channel 4.Output
//     PlcTask Outputs/GVL_iXlinker.EtherCAT_Master_EKxxxx.Beckhoff_EKx9xx.Beckhoff_EKx9xxEK1122.A_0001_EK1960_0000_0019.Module_1_FSoE.FSoE_Outputs.FSOE/FSOUT_Module_6_Channel_1_Output <-> Module 1 (FSoE)/FSoE Outputs/FSOE/FSOUT Module 6.Channel 1.Output
//     PlcTask Outputs/GVL_iXlinker.EtherCAT_Master_EKxxxx.Beckhoff_EKx9xx.Beckhoff_EKx9xxEK1122.A_0001_EK1960_0000_0019.Module_1_FSoE.FSoE_Outputs.FSOE/FSOUT_Module_6_Channel_2_Output <-> Module 1 (FSoE)/FSoE Outputs/FSOE/FSOUT Module 6.Channel 2.Output
//     PlcTask Outputs/GVL_iXlinker.EtherCAT_Master_EKxxxx.Beckhoff_EKx9xx.Beckhoff_EKx9xxEK1122.A_0001_EK1960_0000_0019.Module_1_FSoE.FSoE_Outputs.FSOE/FSOUT_Module_6_Channel_3_Output <-> Module 1 (FSoE)/FSoE Outputs/FSOE/FSOUT Module 6.Channel 3.Output
//     PlcTask Outputs/GVL_iXlinker.EtherCAT_Master_EKxxxx.Beckhoff_EKx9xx.Beckhoff_EKx9xxEK1122.A_0001_EK1960_0000_0019.Module_1_FSoE.FSoE_Outputs.FSOE/FSOUT_Module_6_Channel_4_Output <-> Module 1 (FSoE)/FSoE Outputs/FSOE/FSOUT Module 6.Channel 4.Output
//     PlcTask Outputs/GVL_iXlinker.EtherCAT_Master_EKxxxx.Beckhoff_EKx9xx.Beckhoff_EKx9xxEK1122.A_0001_EK1960_0000_0019.Module_1_FSoE.FSoE_Outputs.FSOE/FSOUT_Module_1_ErrAck <-> Module 1 (FSoE)/FSoE Outputs/FSOE/FSOUT Module 1.ErrAck
//     PlcTask Outputs/GVL_iXlinker.EtherCAT_Master_EKxxxx.Beckhoff_EKx9xx.Beckhoff_EKx9xxEK1122.A_0001_EK1960_0000_0019.Module_1_FSoE.FSoE_Outputs.FSOE/FSOUT_Module_2_ErrAck <-> Module 1 (FSoE)/FSoE Outputs/FSOE/FSOUT Module 2.ErrAck
//     PlcTask Outputs/GVL_iXlinker.EtherCAT_Master_EKxxxx.Beckhoff_EKx9xx.Beckhoff_EKx9xxEK1122.A_0001_EK1960_0000_0019.Module_1_FSoE.FSoE_Outputs.FSOE/FSOUT_Module_3_ErrAck <-> Module 1 (FSoE)/FSoE Outputs/FSOE/FSOUT Module 3.ErrAck
//     PlcTask Outputs/GVL_iXlinker.EtherCAT_Master_EKxxxx.Beckhoff_EKx9xx.Beckhoff_EKx9xxEK1122.A_0001_EK1960_0000_0019.Module_1_FSoE.FSoE_Outputs.FSOE/FSOUT_Module_4_ErrAck <-> Module 1 (FSoE)/FSoE Outputs/FSOE/FSOUT Module 4.ErrAck
//     PlcTask Outputs/GVL_iXlinker.EtherCAT_Master_EKxxxx.Beckhoff_EKx9xx.Beckhoff_EKx9xxEK1122.A_0001_EK1960_0000_0019.Module_1_FSoE.FSoE_Outputs.FSOE/FSOUT_Module_5_ErrAck <-> Module 1 (FSoE)/FSoE Outputs/FSOE/FSOUT Module 5.ErrAck
//     PlcTask Outputs/GVL_iXlinker.EtherCAT_Master_EKxxxx.Beckhoff_EKx9xx.Beckhoff_EKx9xxEK1122.A_0001_EK1960_0000_0019.Module_1_FSoE.FSoE_Outputs.FSOE/FSOUT_Module_6_ErrAck <-> Module 1 (FSoE)/FSoE Outputs/FSOE/FSOUT Module 6.ErrAck
//     PlcTask Outputs/GVL_iXlinker.EtherCAT_Master_EKxxxx.Beckhoff_EKx9xx.Beckhoff_EKx9xxEK1122.A_0001_EK1960_0000_0019.Module_1_FSoE.FSoE_Outputs.FSOE/FSoE_CRC_000 <-> Module 1 (FSoE)/FSoE Outputs/FSOE/FSoE CRC 000
//     PlcTask Outputs/GVL_iXlinker.EtherCAT_Master_EKxxxx.Beckhoff_EKx9xx.Beckhoff_EKx9xxEK1122.A_0001_EK1960_0000_0019.Module_1_FSoE.FSoE_Outputs.FSOE/FSoE_CRC_001 <-> Module 1 (FSoE)/FSoE Outputs/FSOE/FSoE CRC 001
//     PlcTask Outputs/GVL_iXlinker.EtherCAT_Master_EKxxxx.Beckhoff_EKx9xx.Beckhoff_EKx9xxEK1122.A_0001_EK1960_0000_0019.Module_1_FSoE.FSoE_Outputs.FSOE/FSoE_CRC_002 <-> Module 1 (FSoE)/FSoE Outputs/FSOE/FSoE CRC 002
//     PlcTask Outputs/GVL_iXlinker.EtherCAT_Master_EKxxxx.Beckhoff_EKx9xx.Beckhoff_EKx9xxEK1122.A_0001_EK1960_0000_0019.Module_1_FSoE.FSoE_Outputs.FSOE/FSIN_Module_1_ErrAck <-> Module 1 (FSoE)/FSoE Outputs/FSOE/FSIN Module 1.ErrAck
//     PlcTask Outputs/GVL_iXlinker.EtherCAT_Master_EKxxxx.Beckhoff_EKx9xx.Beckhoff_EKx9xxEK1122.A_0001_EK1960_0000_0019.Module_1_FSoE.FSoE_Outputs.FSOE/FSIN_Module_2_ErrAck <-> Module 1 (FSoE)/FSoE Outputs/FSOE/FSIN Module 2.ErrAck
//     PlcTask Outputs/GVL_iXlinker.EtherCAT_Master_EKxxxx.Beckhoff_EKx9xx.Beckhoff_EKx9xxEK1122.A_0001_EK1960_0000_0019.Module_1_FSoE.FSoE_Outputs.FSOE/FSIN_Module_3_ErrAck <-> Module 1 (FSoE)/FSoE Outputs/FSOE/FSIN Module 3.ErrAck
//     PlcTask Outputs/GVL_iXlinker.EtherCAT_Master_EKxxxx.Beckhoff_EKx9xx.Beckhoff_EKx9xxEK1122.A_0001_EK1960_0000_0019.Module_1_FSoE.FSoE_Outputs.FSOE/FSIN_Module_4_ErrAck <-> Module 1 (FSoE)/FSoE Outputs/FSOE/FSIN Module 4.ErrAck
//     PlcTask Outputs/GVL_iXlinker.EtherCAT_Master_EKxxxx.Beckhoff_EKx9xx.Beckhoff_EKx9xxEK1122.A_0001_EK1960_0000_0019.Module_1_FSoE.FSoE_Outputs.FSOE/FSIN_Module_5_ErrAck <-> Module 1 (FSoE)/FSoE Outputs/FSOE/FSIN Module 5.ErrAck
//     PlcTask Outputs/GVL_iXlinker.EtherCAT_Master_EKxxxx.Beckhoff_EKx9xx.Beckhoff_EKx9xxEK1122.A_0001_EK1960_0000_0019.Module_1_FSoE.FSoE_Outputs.FSOE/FSIN_Module_6_ErrAck <-> Module 1 (FSoE)/FSoE Outputs/FSOE/FSIN Module 6.ErrAck
//     PlcTask Outputs/GVL_iXlinker.EtherCAT_Master_EKxxxx.Beckhoff_EKx9xx.Beckhoff_EKx9xxEK1122.A_0001_EK1960_0000_0019.Module_1_FSoE.FSoE_Outputs.FSOE/FSIN_Module_7_ErrAck <-> Module 1 (FSoE)/FSoE Outputs/FSOE/FSIN Module 7.ErrAck
//     PlcTask Outputs/GVL_iXlinker.EtherCAT_Master_EKxxxx.Beckhoff_EKx9xx.Beckhoff_EKx9xxEK1122.A_0001_EK1960_0000_0019.Module_1_FSoE.FSoE_Outputs.FSOE/FSIN_Module_8_ErrAck <-> Module 1 (FSoE)/FSoE Outputs/FSOE/FSIN Module 8.ErrAck
//     PlcTask Outputs/GVL_iXlinker.EtherCAT_Master_EKxxxx.Beckhoff_EKx9xx.Beckhoff_EKx9xxEK1122.A_0001_EK1960_0000_0019.Module_1_FSoE.FSoE_Outputs.FSOE/FSIN_Module_9_ErrAck_1 <-> Module 1 (FSoE)/FSoE Outputs/FSOE/FSIN Module 9.ErrAck 1
//     PlcTask Outputs/GVL_iXlinker.EtherCAT_Master_EKxxxx.Beckhoff_EKx9xx.Beckhoff_EKx9xxEK1122.A_0001_EK1960_0000_0019.Module_1_FSoE.FSoE_Outputs.FSOE/FSIN_Module_9_ErrAck_2 <-> Module 1 (FSoE)/FSoE Outputs/FSOE/FSIN Module 9.ErrAck 2
//     PlcTask Outputs/GVL_iXlinker.EtherCAT_Master_EKxxxx.Beckhoff_EKx9xx.Beckhoff_EKx9xxEK1122.A_0001_EK1960_0000_0019.Module_1_FSoE.FSoE_Outputs.FSOE/FSIN_Module_10_ErrAck_1 <-> Module 1 (FSoE)/FSoE Outputs/FSOE/FSIN Module 10.ErrAck 1
//     PlcTask Outputs/GVL_iXlinker.EtherCAT_Master_EKxxxx.Beckhoff_EKx9xx.Beckhoff_EKx9xxEK1122.A_0001_EK1960_0000_0019.Module_1_FSoE.FSoE_Outputs.FSOE/FSIN_Module_10_ErrAck_2 <-> Module 1 (FSoE)/FSoE Outputs/FSOE/FSIN Module 10.ErrAck 2
//     PlcTask Outputs/GVL_iXlinker.EtherCAT_Master_EKxxxx.Beckhoff_EKx9xx.Beckhoff_EKx9xxEK1122.A_0001_EK1960_0000_0019.Module_1_FSoE.FSoE_Outputs.FSOE/FSoE_Connection_ID <-> Module 1 (FSoE)/FSoE Outputs/FSOE/FSoE Connection ID
//     PlcTask Outputs/GVL_iXlinker.EtherCAT_Master_EKxxxx.Beckhoff_EKx9xx.Beckhoff_EKx9xxEK1122.A_0001_EK1960_0000_0019.Module_2_FSOUT.Outputs.Module_1_Channel_1_Standard_Output_X5_1 <-> Module 2 (FSOUT)/Outputs/Module 1.Channel 1.Standard Output (X5.1)
//     PlcTask Outputs/GVL_iXlinker.EtherCAT_Master_EKxxxx.Beckhoff_EKx9xx.Beckhoff_EKx9xxEK1122.A_0001_EK1960_0000_0019.Module_2_FSOUT.Outputs.Module_1_Channel_2_Standard_Output_X5_2 <-> Module 2 (FSOUT)/Outputs/Module 1.Channel 2.Standard Output (X5.2)
//     PlcTask Outputs/GVL_iXlinker.EtherCAT_Master_EKxxxx.Beckhoff_EKx9xx.Beckhoff_EKx9xxEK1122.A_0001_EK1960_0000_0019.Module_2_FSOUT.Outputs.Module_1_Channel_3_Standard_Output_X5_3 <-> Module 2 (FSOUT)/Outputs/Module 1.Channel 3.Standard Output (X5.3)
//     PlcTask Outputs/GVL_iXlinker.EtherCAT_Master_EKxxxx.Beckhoff_EKx9xx.Beckhoff_EKx9xxEK1122.A_0001_EK1960_0000_0019.Module_2_FSOUT.Outputs.Module_1_Channel_4_Standard_Output_X5_4 <-> Module 2 (FSOUT)/Outputs/Module 1.Channel 4.Standard Output (X5.4)
//     PlcTask Outputs/GVL_iXlinker.EtherCAT_Master_EKxxxx.Beckhoff_EKx9xx.Beckhoff_EKx9xxEK1122.A_0001_EK1960_0000_0019.Module_2_FSOUT.Outputs.Module_2_Channel_1_Standard_Output_X5_5 <-> Module 2 (FSOUT)/Outputs/Module 2.Channel 1.Standard Output (X5.5)
//     PlcTask Outputs/GVL_iXlinker.EtherCAT_Master_EKxxxx.Beckhoff_EKx9xx.Beckhoff_EKx9xxEK1122.A_0001_EK1960_0000_0019.Module_2_FSOUT.Outputs.Module_2_Channel_2_Standard_Output_X5_6 <-> Module 2 (FSOUT)/Outputs/Module 2.Channel 2.Standard Output (X5.6)
//     PlcTask Outputs/GVL_iXlinker.EtherCAT_Master_EKxxxx.Beckhoff_EKx9xx.Beckhoff_EKx9xxEK1122.A_0001_EK1960_0000_0019.Module_2_FSOUT.Outputs.Module_2_Channel_3_Standard_Output_X5_7 <-> Module 2 (FSOUT)/Outputs/Module 2.Channel 3.Standard Output (X5.7)
//     PlcTask Outputs/GVL_iXlinker.EtherCAT_Master_EKxxxx.Beckhoff_EKx9xx.Beckhoff_EKx9xxEK1122.A_0001_EK1960_0000_0019.Module_2_FSOUT.Outputs.Module_2_Channel_4_Standard_Output_X5_8 <-> Module 2 (FSOUT)/Outputs/Module 2.Channel 4.Standard Output (X5.8)
//     PlcTask Outputs/GVL_iXlinker.EtherCAT_Master_EKxxxx.Beckhoff_EKx9xx.Beckhoff_EKx9xxEK1122.A_0001_EK1960_0000_0019.Module_2_FSOUT.Outputs.Module_3_Channel_1_Standard_Output_X7_1 <-> Module 2 (FSOUT)/Outputs/Module 3.Channel 1.Standard Output (X7.1)
//     PlcTask Outputs/GVL_iXlinker.EtherCAT_Master_EKxxxx.Beckhoff_EKx9xx.Beckhoff_EKx9xxEK1122.A_0001_EK1960_0000_0019.Module_2_FSOUT.Outputs.Module_3_Channel_2_Standard_Output_X7_2 <-> Module 2 (FSOUT)/Outputs/Module 3.Channel 2.Standard Output (X7.2)
//     PlcTask Outputs/GVL_iXlinker.EtherCAT_Master_EKxxxx.Beckhoff_EKx9xx.Beckhoff_EKx9xxEK1122.A_0001_EK1960_0000_0019.Module_2_FSOUT.Outputs.Module_3_Channel_3_Standard_Output_X7_3 <-> Module 2 (FSOUT)/Outputs/Module 3.Channel 3.Standard Output (X7.3)
//     PlcTask Outputs/GVL_iXlinker.EtherCAT_Master_EKxxxx.Beckhoff_EKx9xx.Beckhoff_EKx9xxEK1122.A_0001_EK1960_0000_0019.Module_2_FSOUT.Outputs.Module_3_Channel_4_Standard_Output_X7_4 <-> Module 2 (FSOUT)/Outputs/Module 3.Channel 4.Standard Output (X7.4)
//     PlcTask Outputs/GVL_iXlinker.EtherCAT_Master_EKxxxx.Beckhoff_EKx9xx.Beckhoff_EKx9xxEK1122.A_0001_EK1960_0000_0019.Module_2_FSOUT.Outputs.Module_4_Channel_1_Standard_Output_X7_5 <-> Module 2 (FSOUT)/Outputs/Module 4.Channel 1.Standard Output (X7.5)
//     PlcTask Outputs/GVL_iXlinker.EtherCAT_Master_EKxxxx.Beckhoff_EKx9xx.Beckhoff_EKx9xxEK1122.A_0001_EK1960_0000_0019.Module_2_FSOUT.Outputs.Module_4_Channel_2_Standard_Output_X7_6 <-> Module 2 (FSOUT)/Outputs/Module 4.Channel 2.Standard Output (X7.6)
//     PlcTask Outputs/GVL_iXlinker.EtherCAT_Master_EKxxxx.Beckhoff_EKx9xx.Beckhoff_EKx9xxEK1122.A_0001_EK1960_0000_0019.Module_2_FSOUT.Outputs.Module_4_Channel_3_Standard_Output_X7_7 <-> Module 2 (FSOUT)/Outputs/Module 4.Channel 3.Standard Output (X7.7)
//     PlcTask Outputs/GVL_iXlinker.EtherCAT_Master_EKxxxx.Beckhoff_EKx9xx.Beckhoff_EKx9xxEK1122.A_0001_EK1960_0000_0019.Module_2_FSOUT.Outputs.Module_4_Channel_4_Standard_Output_X7_8 <-> Module 2 (FSOUT)/Outputs/Module 4.Channel 4.Standard Output (X7.8)
//     PlcTask Outputs/GVL_iXlinker.EtherCAT_Master_EKxxxx.Beckhoff_EKx9xx.Beckhoff_EKx9xxEK1122.A_0001_EK1960_0000_0019.Module_2_FSOUT.Outputs.Module_5_Channel_1_Standard_Output_X9_1 <-> Module 2 (FSOUT)/Outputs/Module 5.Channel 1.Standard Output (X9.1)
//     PlcTask Outputs/GVL_iXlinker.EtherCAT_Master_EKxxxx.Beckhoff_EKx9xx.Beckhoff_EKx9xxEK1122.A_0001_EK1960_0000_0019.Module_2_FSOUT.Outputs.Module_5_Channel_2_Standard_Output_X9_2 <-> Module 2 (FSOUT)/Outputs/Module 5.Channel 2.Standard Output (X9.2)
//     PlcTask Outputs/GVL_iXlinker.EtherCAT_Master_EKxxxx.Beckhoff_EKx9xx.Beckhoff_EKx9xxEK1122.A_0001_EK1960_0000_0019.Module_2_FSOUT.Outputs.Module_5_Channel_3_Standard_Output_X9_3 <-> Module 2 (FSOUT)/Outputs/Module 5.Channel 3.Standard Output (X9.3)
//     PlcTask Outputs/GVL_iXlinker.EtherCAT_Master_EKxxxx.Beckhoff_EKx9xx.Beckhoff_EKx9xxEK1122.A_0001_EK1960_0000_0019.Module_2_FSOUT.Outputs.Module_5_Channel_4_Standard_Output_X9_4 <-> Module 2 (FSOUT)/Outputs/Module 5.Channel 4.Standard Output (X9.4)
//     PlcTask Outputs/GVL_iXlinker.EtherCAT_Master_EKxxxx.Beckhoff_EKx9xx.Beckhoff_EKx9xxEK1122.A_0001_EK1960_0000_0019.Module_2_FSOUT.Outputs.Module_6_Channel_1_Standard_Output_X9_5 <-> Module 2 (FSOUT)/Outputs/Module 6.Channel 1.Standard Output (X9.5)
//     PlcTask Outputs/GVL_iXlinker.EtherCAT_Master_EKxxxx.Beckhoff_EKx9xx.Beckhoff_EKx9xxEK1122.A_0001_EK1960_0000_0019.Module_2_FSOUT.Outputs.Module_6_Channel_2_Standard_Output_X9_6 <-> Module 2 (FSOUT)/Outputs/Module 6.Channel 2.Standard Output (X9.6)
//     PlcTask Outputs/GVL_iXlinker.EtherCAT_Master_EKxxxx.Beckhoff_EKx9xx.Beckhoff_EKx9xxEK1122.A_0001_EK1960_0000_0019.Module_2_FSOUT.Outputs.Module_6_Channel_3_Standard_Output_X9_7 <-> Module 2 (FSOUT)/Outputs/Module 6.Channel 3.Standard Output (X9.7)
//     PlcTask Outputs/GVL_iXlinker.EtherCAT_Master_EKxxxx.Beckhoff_EKx9xx.Beckhoff_EKx9xxEK1122.A_0001_EK1960_0000_0019.Module_2_FSOUT.Outputs.Module_6_Channel_4_Standard_Output_X9_8 <-> Module 2 (FSOUT)/Outputs/Module 6.Channel 4.Standard Output (X9.8)
//     PlcTask Outputs/GVL_iXlinker.EtherCAT_Master_EKxxxx.Beckhoff_EKx9xx.Beckhoff_EKx9xxEK1122.A_0001_EK1960_0000_0019.Module_2_FSOUT.Outputs.Relais_Module_Channel_1_Standard_Output_X4_1_X4_5 <-> Module 2 (FSOUT)/Outputs/Relais Module.Channel 1.Standard Output (X4.1, X4.5)
//     PlcTask Outputs/GVL_iXlinker.EtherCAT_Master_EKxxxx.Beckhoff_EKx9xx.Beckhoff_EKx9xxEK1122.A_0001_EK1960_0000_0019.Module_2_FSOUT.Outputs.Relais_Module_Channel_2_Standard_Output_X4_2_X4_6 <-> Module 2 (FSOUT)/Outputs/Relais Module.Channel 2.Standard Output (X4.2, X4.6)
//     PlcTask Outputs/GVL_iXlinker.EtherCAT_Master_EKxxxx.Beckhoff_EKx9xx.Beckhoff_EKx9xxEK1122.A_0001_EK1960_0000_0019.Module_2_FSOUT.Outputs.Relais_Module_Channel_3_Standard_Output_X4_3_X4_7 <-> Module 2 (FSOUT)/Outputs/Relais Module.Channel 3.Standard Output (X4.3, X4.7)
//     PlcTask Outputs/GVL_iXlinker.EtherCAT_Master_EKxxxx.Beckhoff_EKx9xx.Beckhoff_EKx9xxEK1122.A_0001_EK1960_0000_0019.Module_2_FSOUT.Outputs.Relais_Module_Channel_4_Standard_Output_X4_4_X4_8 <-> Module 2 (FSOUT)/Outputs/Relais Module.Channel 4.Standard Output (X4.4, X4.8)
//     PlcTask Inputs/GVL_iXlinker.EtherCAT_Master_EKxxxx.Beckhoff_EKx9xx.Beckhoff_EKx9xxEK1122.A_0001_EK1960_0000_0019.Module_3_FSLOGIC.FSLOGIC_Inputs.Safe_Logic_State <-> Module 3 (FSLOGIC)/FSLOGIC Inputs/Safe Logic State
//     PlcTask Inputs/GVL_iXlinker.EtherCAT_Master_EKxxxx.Beckhoff_EKx9xx.Beckhoff_EKx9xxEK1122.A_0001_EK1960_0000_0019.Module_3_FSLOGIC.FSLOGIC_Inputs.Cycle_Counter <-> Module 3 (FSLOGIC)/FSLOGIC Inputs/Cycle Counter
//     PlcTask Inputs/GVL_iXlinker.EtherCAT_Master_EKxxxx.Beckhoff_EKx9xx.Beckhoff_EKx9xxEK1122.A_0001_EK1960_0000_0019.WcState.WcState0 <-> WcState/WcState0
//     PlcTask Inputs/GVL_iXlinker.EtherCAT_Master_EKxxxx.Beckhoff_EKx9xx.Beckhoff_EKx9xxEK1122.A_0001_EK1960_0000_0019.WcState.WcState1 <-> WcState/WcState1
//     PlcTask Inputs/GVL_iXlinker.EtherCAT_Master_EKxxxx.Beckhoff_EKx9xx.Beckhoff_EKx9xxEK1122.A_0001_EK1960_0000_0019.WcState.InputToggle0 <-> WcState/InputToggle0
//     PlcTask Inputs/GVL_iXlinker.EtherCAT_Master_EKxxxx.Beckhoff_EKx9xx.Beckhoff_EKx9xxEK1122.A_0001_EK1960_0000_0019.WcState.InputToggle1 <-> WcState/InputToggle1
//     PlcTask Inputs/GVL_iXlinker.EtherCAT_Master_EKxxxx.Beckhoff_EKx9xx.Beckhoff_EKx9xxEK1122.A_0001_EK1960_0000_0019.InfoData.AdsAddr <-> InfoData/AdsAddr
//     PlcTask Inputs/GVL_iXlinker.EtherCAT_Master_EKxxxx.Beckhoff_EKx9xx.Beckhoff_EKx9xxEK1122.A_0001_EK1960_0000_0019.InfoData.State <-> InfoData/State
//   PLC/PLC Instance <-> EtherCAT Master EKxxxx/Beckhoff EKx9xx/Beckhoff EKx9xxEK1122/A_0002(EK1960-0000-0021)
//     PlcTask Inputs/GVL_iXlinker.EtherCAT_Master_EKxxxx.Beckhoff_EKx9xx.Beckhoff_EKx9xxEK1122.A_0002_EK1960_0000_0021.Module_1_FSoE.FSoE_Inputs.FSOE/FSoE_Command <-> Module 1 (FSoE)/FSoE Inputs/FSOE/FSoE Command
//     PlcTask Inputs/GVL_iXlinker.EtherCAT_Master_EKxxxx.Beckhoff_EKx9xx.Beckhoff_EKx9xxEK1122.A_0002_EK1960_0000_0021.Module_1_FSoE.FSoE_Inputs.FSOE/FSOUT_Module_1_Module_Fault <-> Module 1 (FSoE)/FSoE Inputs/FSOE/FSOUT Module 1.Module Fault
//     PlcTask Inputs/GVL_iXlinker.EtherCAT_Master_EKxxxx.Beckhoff_EKx9xx.Beckhoff_EKx9xxEK1122.A_0002_EK1960_0000_0021.Module_1_FSoE.FSoE_Inputs.FSOE/FSOUT_Module_2_Module_Fault <-> Module 1 (FSoE)/FSoE Inputs/FSOE/FSOUT Module 2.Module Fault
//     PlcTask Inputs/GVL_iXlinker.EtherCAT_Master_EKxxxx.Beckhoff_EKx9xx.Beckhoff_EKx9xxEK1122.A_0002_EK1960_0000_0021.Module_1_FSoE.FSoE_Inputs.FSOE/FSOUT_Module_3_Module_Fault <-> Module 1 (FSoE)/FSoE Inputs/FSOE/FSOUT Module 3.Module Fault
//     PlcTask Inputs/GVL_iXlinker.EtherCAT_Master_EKxxxx.Beckhoff_EKx9xx.Beckhoff_EKx9xxEK1122.A_0002_EK1960_0000_0021.Module_1_FSoE.FSoE_Inputs.FSOE/FSOUT_Module_4_Module_Fault <-> Module 1 (FSoE)/FSoE Inputs/FSOE/FSOUT Module 4.Module Fault
//     PlcTask Inputs/GVL_iXlinker.EtherCAT_Master_EKxxxx.Beckhoff_EKx9xx.Beckhoff_EKx9xxEK1122.A_0002_EK1960_0000_0021.Module_1_FSoE.FSoE_Inputs.FSOE/FSOUT_Module_5_Module_Fault <-> Module 1 (FSoE)/FSoE Inputs/FSOE/FSOUT Module 5.Module Fault
//     PlcTask Inputs/GVL_iXlinker.EtherCAT_Master_EKxxxx.Beckhoff_EKx9xx.Beckhoff_EKx9xxEK1122.A_0002_EK1960_0000_0021.Module_1_FSoE.FSoE_Inputs.FSOE/FSOUT_Module_6_Module_Fault <-> Module 1 (FSoE)/FSoE Inputs/FSOE/FSOUT Module 6.Module Fault
//     PlcTask Inputs/GVL_iXlinker.EtherCAT_Master_EKxxxx.Beckhoff_EKx9xx.Beckhoff_EKx9xxEK1122.A_0002_EK1960_0000_0021.Module_1_FSoE.FSoE_Inputs.FSOE/FSIN_Module_1_Channel_1_Input_X6_1 <-> Module 1 (FSoE)/FSoE Inputs/FSOE/FSIN Module 1.Channel 1.Input (X6.1)
//     PlcTask Inputs/GVL_iXlinker.EtherCAT_Master_EKxxxx.Beckhoff_EKx9xx.Beckhoff_EKx9xxEK1122.A_0002_EK1960_0000_0021.Module_1_FSoE.FSoE_Inputs.FSOE/FSIN_Module_1_Channel_2_Input_X6_2 <-> Module 1 (FSoE)/FSoE Inputs/FSOE/FSIN Module 1.Channel 2.Input (X6.2)
//     PlcTask Inputs/GVL_iXlinker.EtherCAT_Master_EKxxxx.Beckhoff_EKx9xx.Beckhoff_EKx9xxEK1122.A_0002_EK1960_0000_0021.Module_1_FSoE.FSoE_Inputs.FSOE/FSIN_Module_2_Channel_1_Input_X6_3 <-> Module 1 (FSoE)/FSoE Inputs/FSOE/FSIN Module 2.Channel 1.Input (X6.3)
//     PlcTask Inputs/GVL_iXlinker.EtherCAT_Master_EKxxxx.Beckhoff_EKx9xx.Beckhoff_EKx9xxEK1122.A_0002_EK1960_0000_0021.Module_1_FSoE.FSoE_Inputs.FSOE/FSIN_Module_2_Channel_2_Input_X6_4 <-> Module 1 (FSoE)/FSoE Inputs/FSOE/FSIN Module 2.Channel 2.Input (X6.4)
//     PlcTask Inputs/GVL_iXlinker.EtherCAT_Master_EKxxxx.Beckhoff_EKx9xx.Beckhoff_EKx9xxEK1122.A_0002_EK1960_0000_0021.Module_1_FSoE.FSoE_Inputs.FSOE/FSIN_Module_3_Channel_1_Input_X6_5 <-> Module 1 (FSoE)/FSoE Inputs/FSOE/FSIN Module 3.Channel 1.Input (X6.5)
//     PlcTask Inputs/GVL_iXlinker.EtherCAT_Master_EKxxxx.Beckhoff_EKx9xx.Beckhoff_EKx9xxEK1122.A_0002_EK1960_0000_0021.Module_1_FSoE.FSoE_Inputs.FSOE/FSIN_Module_3_Channel_2_Input_X6_6 <-> Module 1 (FSoE)/FSoE Inputs/FSOE/FSIN Module 3.Channel 2.Input (X6.6)
//     PlcTask Inputs/GVL_iXlinker.EtherCAT_Master_EKxxxx.Beckhoff_EKx9xx.Beckhoff_EKx9xxEK1122.A_0002_EK1960_0000_0021.Module_1_FSoE.FSoE_Inputs.FSOE/FSIN_Module_4_Channel_1_Input_X6_7 <-> Module 1 (FSoE)/FSoE Inputs/FSOE/FSIN Module 4.Channel 1.Input (X6.7)
//     PlcTask Inputs/GVL_iXlinker.EtherCAT_Master_EKxxxx.Beckhoff_EKx9xx.Beckhoff_EKx9xxEK1122.A_0002_EK1960_0000_0021.Module_1_FSoE.FSoE_Inputs.FSOE/FSIN_Module_4_Channel_2_Input_X6_8 <-> Module 1 (FSoE)/FSoE Inputs/FSOE/FSIN Module 4.Channel 2.Input (X6.8)
//     PlcTask Inputs/GVL_iXlinker.EtherCAT_Master_EKxxxx.Beckhoff_EKx9xx.Beckhoff_EKx9xxEK1122.A_0002_EK1960_0000_0021.Module_1_FSoE.FSoE_Inputs.FSOE/FSIN_Module_5_Channel_1_Input_X6_9 <-> Module 1 (FSoE)/FSoE Inputs/FSOE/FSIN Module 5.Channel 1.Input (X6.9)
//     PlcTask Inputs/GVL_iXlinker.EtherCAT_Master_EKxxxx.Beckhoff_EKx9xx.Beckhoff_EKx9xxEK1122.A_0002_EK1960_0000_0021.Module_1_FSoE.FSoE_Inputs.FSOE/FSIN_Module_5_Channel_2_Input_X6_10 <-> Module 1 (FSoE)/FSoE Inputs/FSOE/FSIN Module 5.Channel 2.Input (X6.10)
//     PlcTask Inputs/GVL_iXlinker.EtherCAT_Master_EKxxxx.Beckhoff_EKx9xx.Beckhoff_EKx9xxEK1122.A_0002_EK1960_0000_0021.Module_1_FSoE.FSoE_Inputs.FSOE/FSIN_Module_6_Channel_1_Input_X8_1 <-> Module 1 (FSoE)/FSoE Inputs/FSOE/FSIN Module 6.Channel 1.Input (X8.1)
//     PlcTask Inputs/GVL_iXlinker.EtherCAT_Master_EKxxxx.Beckhoff_EKx9xx.Beckhoff_EKx9xxEK1122.A_0002_EK1960_0000_0021.Module_1_FSoE.FSoE_Inputs.FSOE/FSIN_Module_6_Channel_2_Input_X8_2 <-> Module 1 (FSoE)/FSoE Inputs/FSOE/FSIN Module 6.Channel 2.Input (X8.2)
//     PlcTask Inputs/GVL_iXlinker.EtherCAT_Master_EKxxxx.Beckhoff_EKx9xx.Beckhoff_EKx9xxEK1122.A_0002_EK1960_0000_0021.Module_1_FSoE.FSoE_Inputs.FSOE/FSIN_Module_7_Channel_1_Input_X8_3 <-> Module 1 (FSoE)/FSoE Inputs/FSOE/FSIN Module 7.Channel 1.Input (X8.3)
//     PlcTask Inputs/GVL_iXlinker.EtherCAT_Master_EKxxxx.Beckhoff_EKx9xx.Beckhoff_EKx9xxEK1122.A_0002_EK1960_0000_0021.Module_1_FSoE.FSoE_Inputs.FSOE/FSIN_Module_7_Channel_2_Input_X8_4 <-> Module 1 (FSoE)/FSoE Inputs/FSOE/FSIN Module 7.Channel 2.Input (X8.4)
//     PlcTask Inputs/GVL_iXlinker.EtherCAT_Master_EKxxxx.Beckhoff_EKx9xx.Beckhoff_EKx9xxEK1122.A_0002_EK1960_0000_0021.Module_1_FSoE.FSoE_Inputs.FSOE/FSIN_Module_8_Channel_1_Input_X8_5 <-> Module 1 (FSoE)/FSoE Inputs/FSOE/FSIN Module 8.Channel 1.Input (X8.5)
//     PlcTask Inputs/GVL_iXlinker.EtherCAT_Master_EKxxxx.Beckhoff_EKx9xx.Beckhoff_EKx9xxEK1122.A_0002_EK1960_0000_0021.Module_1_FSoE.FSoE_Inputs.FSOE/FSIN_Module_8_Channel_2_Input_X8_6 <-> Module 1 (FSoE)/FSoE Inputs/FSOE/FSIN Module 8.Channel 2.Input (X8.6)
//     PlcTask Inputs/GVL_iXlinker.EtherCAT_Master_EKxxxx.Beckhoff_EKx9xx.Beckhoff_EKx9xxEK1122.A_0002_EK1960_0000_0021.Module_1_FSoE.FSoE_Inputs.FSOE/FSIN_Module_9_Channel_1_Input_X8_7 <-> Module 1 (FSoE)/FSoE Inputs/FSOE/FSIN Module 9.Channel 1.Input (X8.7)
//     PlcTask Inputs/GVL_iXlinker.EtherCAT_Master_EKxxxx.Beckhoff_EKx9xx.Beckhoff_EKx9xxEK1122.A_0002_EK1960_0000_0021.Module_1_FSoE.FSoE_Inputs.FSOE/FSIN_Module_9_Channel_2_Input_X8_8 <-> Module 1 (FSoE)/FSoE Inputs/FSOE/FSIN Module 9.Channel 2.Input (X8.8)
//     PlcTask Inputs/GVL_iXlinker.EtherCAT_Master_EKxxxx.Beckhoff_EKx9xx.Beckhoff_EKx9xxEK1122.A_0002_EK1960_0000_0021.Module_1_FSoE.FSoE_Inputs.FSOE/FSIN_Module_10_Channel_1_Input_X8_9 <-> Module 1 (FSoE)/FSoE Inputs/FSOE/FSIN Module 10.Channel 1.Input (X8.9)
//     PlcTask Inputs/GVL_iXlinker.EtherCAT_Master_EKxxxx.Beckhoff_EKx9xx.Beckhoff_EKx9xxEK1122.A_0002_EK1960_0000_0021.Module_1_FSoE.FSoE_Inputs.FSOE/FSIN_Module_10_Channel_2_Input_X8_10 <-> Module 1 (FSoE)/FSoE Inputs/FSOE/FSIN Module 10.Channel 2.Input (X8.10)
//     PlcTask Inputs/GVL_iXlinker.EtherCAT_Master_EKxxxx.Beckhoff_EKx9xx.Beckhoff_EKx9xxEK1122.A_0002_EK1960_0000_0021.Module_1_FSoE.FSoE_Inputs.FSOE/FSIN_Module_1_Module_Fault <-> Module 1 (FSoE)/FSoE Inputs/FSOE/FSIN Module 1.Module Fault
//     PlcTask Inputs/GVL_iXlinker.EtherCAT_Master_EKxxxx.Beckhoff_EKx9xx.Beckhoff_EKx9xxEK1122.A_0002_EK1960_0000_0021.Module_1_FSoE.FSoE_Inputs.FSOE/FSIN_Module_2_Module_Fault <-> Module 1 (FSoE)/FSoE Inputs/FSOE/FSIN Module 2.Module Fault
//     PlcTask Inputs/GVL_iXlinker.EtherCAT_Master_EKxxxx.Beckhoff_EKx9xx.Beckhoff_EKx9xxEK1122.A_0002_EK1960_0000_0021.Module_1_FSoE.FSoE_Inputs.FSOE/FSIN_Module_3_Module_Fault <-> Module 1 (FSoE)/FSoE Inputs/FSOE/FSIN Module 3.Module Fault
//     PlcTask Inputs/GVL_iXlinker.EtherCAT_Master_EKxxxx.Beckhoff_EKx9xx.Beckhoff_EKx9xxEK1122.A_0002_EK1960_0000_0021.Module_1_FSoE.FSoE_Inputs.FSOE/FSIN_Module_4_Module_Fault <-> Module 1 (FSoE)/FSoE Inputs/FSOE/FSIN Module 4.Module Fault
//     PlcTask Inputs/GVL_iXlinker.EtherCAT_Master_EKxxxx.Beckhoff_EKx9xx.Beckhoff_EKx9xxEK1122.A_0002_EK1960_0000_0021.Module_1_FSoE.FSoE_Inputs.FSOE/FSIN_Module_5_Module_Fault <-> Module 1 (FSoE)/FSoE Inputs/FSOE/FSIN Module 5.Module Fault
//     PlcTask Inputs/GVL_iXlinker.EtherCAT_Master_EKxxxx.Beckhoff_EKx9xx.Beckhoff_EKx9xxEK1122.A_0002_EK1960_0000_0021.Module_1_FSoE.FSoE_Inputs.FSOE/FSIN_Module_6_Module_Fault <-> Module 1 (FSoE)/FSoE Inputs/FSOE/FSIN Module 6.Module Fault
//     PlcTask Inputs/GVL_iXlinker.EtherCAT_Master_EKxxxx.Beckhoff_EKx9xx.Beckhoff_EKx9xxEK1122.A_0002_EK1960_0000_0021.Module_1_FSoE.FSoE_Inputs.FSOE/FSIN_Module_7_Module_Fault <-> Module 1 (FSoE)/FSoE Inputs/FSOE/FSIN Module 7.Module Fault
//     PlcTask Inputs/GVL_iXlinker.EtherCAT_Master_EKxxxx.Beckhoff_EKx9xx.Beckhoff_EKx9xxEK1122.A_0002_EK1960_0000_0021.Module_1_FSoE.FSoE_Inputs.FSOE/FSIN_Module_8_Module_Fault <-> Module 1 (FSoE)/FSoE Inputs/FSOE/FSIN Module 8.Module Fault
//     PlcTask Inputs/GVL_iXlinker.EtherCAT_Master_EKxxxx.Beckhoff_EKx9xx.Beckhoff_EKx9xxEK1122.A_0002_EK1960_0000_0021.Module_1_FSoE.FSoE_Inputs.FSOE/FSoE_CRC_000 <-> Module 1 (FSoE)/FSoE Inputs/FSOE/FSoE CRC 000
//     PlcTask Inputs/GVL_iXlinker.EtherCAT_Master_EKxxxx.Beckhoff_EKx9xx.Beckhoff_EKx9xxEK1122.A_0002_EK1960_0000_0021.Module_1_FSoE.FSoE_Inputs.FSOE/FSoE_CRC_001 <-> Module 1 (FSoE)/FSoE Inputs/FSOE/FSoE CRC 001
//     PlcTask Inputs/GVL_iXlinker.EtherCAT_Master_EKxxxx.Beckhoff_EKx9xx.Beckhoff_EKx9xxEK1122.A_0002_EK1960_0000_0021.Module_1_FSoE.FSoE_Inputs.FSOE/FSoE_CRC_002 <-> Module 1 (FSoE)/FSoE Inputs/FSOE/FSoE CRC 002
//     PlcTask Inputs/GVL_iXlinker.EtherCAT_Master_EKxxxx.Beckhoff_EKx9xx.Beckhoff_EKx9xxEK1122.A_0002_EK1960_0000_0021.Module_1_FSoE.FSoE_Inputs.FSOE/FSIN_Module_9_Module_Fault_1 <-> Module 1 (FSoE)/FSoE Inputs/FSOE/FSIN Module 9.Module Fault 1
//     PlcTask Inputs/GVL_iXlinker.EtherCAT_Master_EKxxxx.Beckhoff_EKx9xx.Beckhoff_EKx9xxEK1122.A_0002_EK1960_0000_0021.Module_1_FSoE.FSoE_Inputs.FSOE/FSIN_Module_9_Module_Fault_2 <-> Module 1 (FSoE)/FSoE Inputs/FSOE/FSIN Module 9.Module Fault 2
//     PlcTask Inputs/GVL_iXlinker.EtherCAT_Master_EKxxxx.Beckhoff_EKx9xx.Beckhoff_EKx9xxEK1122.A_0002_EK1960_0000_0021.Module_1_FSoE.FSoE_Inputs.FSOE/FSIN_Module_10_Module_Fault_1 <-> Module 1 (FSoE)/FSoE Inputs/FSOE/FSIN Module 10.Module Fault 1
//     PlcTask Inputs/GVL_iXlinker.EtherCAT_Master_EKxxxx.Beckhoff_EKx9xx.Beckhoff_EKx9xxEK1122.A_0002_EK1960_0000_0021.Module_1_FSoE.FSoE_Inputs.FSOE/FSIN_Module_10_Module_Fault_2 <-> Module 1 (FSoE)/FSoE Inputs/FSOE/FSIN Module 10.Module Fault 2
//     PlcTask Inputs/GVL_iXlinker.EtherCAT_Master_EKxxxx.Beckhoff_EKx9xx.Beckhoff_EKx9xxEK1122.A_0002_EK1960_0000_0021.Module_1_FSoE.FSoE_Inputs.FSOE/FSoE_Connection_ID <-> Module 1 (FSoE)/FSoE Inputs/FSOE/FSoE Connection ID
//     PlcTask Outputs/GVL_iXlinker.EtherCAT_Master_EKxxxx.Beckhoff_EKx9xx.Beckhoff_EKx9xxEK1122.A_0002_EK1960_0000_0021.Module_1_FSoE.FSoE_Outputs.FSOE/FSoE_Command <-> Module 1 (FSoE)/FSoE Outputs/FSOE/FSoE Command
//     PlcTask Outputs/GVL_iXlinker.EtherCAT_Master_EKxxxx.Beckhoff_EKx9xx.Beckhoff_EKx9xxEK1122.A_0002_EK1960_0000_0021.Module_1_FSoE.FSoE_Outputs.FSOE/FSOUT_Module_1_Channel_1_Output_X5_1 <-> Module 1 (FSoE)/FSoE Outputs/FSOE/FSOUT Module 1.Channel 1.Output (X5.1)
//     PlcTask Outputs/GVL_iXlinker.EtherCAT_Master_EKxxxx.Beckhoff_EKx9xx.Beckhoff_EKx9xxEK1122.A_0002_EK1960_0000_0021.Module_1_FSoE.FSoE_Outputs.FSOE/FSOUT_Module_1_Channel_2_Output_X5_2 <-> Module 1 (FSoE)/FSoE Outputs/FSOE/FSOUT Module 1.Channel 2.Output (X5.2)
//     PlcTask Outputs/GVL_iXlinker.EtherCAT_Master_EKxxxx.Beckhoff_EKx9xx.Beckhoff_EKx9xxEK1122.A_0002_EK1960_0000_0021.Module_1_FSoE.FSoE_Outputs.FSOE/FSOUT_Module_1_Channel_3_Output_X5_3 <-> Module 1 (FSoE)/FSoE Outputs/FSOE/FSOUT Module 1.Channel 3.Output (X5.3)
//     PlcTask Outputs/GVL_iXlinker.EtherCAT_Master_EKxxxx.Beckhoff_EKx9xx.Beckhoff_EKx9xxEK1122.A_0002_EK1960_0000_0021.Module_1_FSoE.FSoE_Outputs.FSOE/FSOUT_Module_1_Channel_4_Output_X5_4 <-> Module 1 (FSoE)/FSoE Outputs/FSOE/FSOUT Module 1.Channel 4.Output (X5.4)
//     PlcTask Outputs/GVL_iXlinker.EtherCAT_Master_EKxxxx.Beckhoff_EKx9xx.Beckhoff_EKx9xxEK1122.A_0002_EK1960_0000_0021.Module_1_FSoE.FSoE_Outputs.FSOE/FSOUT_Module_2_Channel_1_Output_X5_5 <-> Module 1 (FSoE)/FSoE Outputs/FSOE/FSOUT Module 2.Channel 1.Output (X5.5)
//     PlcTask Outputs/GVL_iXlinker.EtherCAT_Master_EKxxxx.Beckhoff_EKx9xx.Beckhoff_EKx9xxEK1122.A_0002_EK1960_0000_0021.Module_1_FSoE.FSoE_Outputs.FSOE/FSOUT_Module_2_Channel_2_Output_X5_6 <-> Module 1 (FSoE)/FSoE Outputs/FSOE/FSOUT Module 2.Channel 2.Output (X5.6)
//     PlcTask Outputs/GVL_iXlinker.EtherCAT_Master_EKxxxx.Beckhoff_EKx9xx.Beckhoff_EKx9xxEK1122.A_0002_EK1960_0000_0021.Module_1_FSoE.FSoE_Outputs.FSOE/FSOUT_Module_2_Channel_3_Output_X5_7 <-> Module 1 (FSoE)/FSoE Outputs/FSOE/FSOUT Module 2.Channel 3.Output (X5.7)
//     PlcTask Outputs/GVL_iXlinker.EtherCAT_Master_EKxxxx.Beckhoff_EKx9xx.Beckhoff_EKx9xxEK1122.A_0002_EK1960_0000_0021.Module_1_FSoE.FSoE_Outputs.FSOE/FSOUT_Module_2_Channel_4_Output_X5_8 <-> Module 1 (FSoE)/FSoE Outputs/FSOE/FSOUT Module 2.Channel 4.Output (X5.8)
//     PlcTask Outputs/GVL_iXlinker.EtherCAT_Master_EKxxxx.Beckhoff_EKx9xx.Beckhoff_EKx9xxEK1122.A_0002_EK1960_0000_0021.Module_1_FSoE.FSoE_Outputs.FSOE/FSOUT_Module_3_Channel_1_Output_X7_1 <-> Module 1 (FSoE)/FSoE Outputs/FSOE/FSOUT Module 3.Channel 1.Output (X7.1)
//     PlcTask Outputs/GVL_iXlinker.EtherCAT_Master_EKxxxx.Beckhoff_EKx9xx.Beckhoff_EKx9xxEK1122.A_0002_EK1960_0000_0021.Module_1_FSoE.FSoE_Outputs.FSOE/FSOUT_Module_3_Channel_2_Output_X7_2 <-> Module 1 (FSoE)/FSoE Outputs/FSOE/FSOUT Module 3.Channel 2.Output (X7.2)
//     PlcTask Outputs/GVL_iXlinker.EtherCAT_Master_EKxxxx.Beckhoff_EKx9xx.Beckhoff_EKx9xxEK1122.A_0002_EK1960_0000_0021.Module_1_FSoE.FSoE_Outputs.FSOE/FSOUT_Module_3_Channel_3_Output_X7_3 <-> Module 1 (FSoE)/FSoE Outputs/FSOE/FSOUT Module 3.Channel 3.Output (X7.3)
//     PlcTask Outputs/GVL_iXlinker.EtherCAT_Master_EKxxxx.Beckhoff_EKx9xx.Beckhoff_EKx9xxEK1122.A_0002_EK1960_0000_0021.Module_1_FSoE.FSoE_Outputs.FSOE/FSOUT_Module_3_Channel_4_Output_X7_4 <-> Module 1 (FSoE)/FSoE Outputs/FSOE/FSOUT Module 3.Channel 4.Output (X7.4)
//     PlcTask Outputs/GVL_iXlinker.EtherCAT_Master_EKxxxx.Beckhoff_EKx9xx.Beckhoff_EKx9xxEK1122.A_0002_EK1960_0000_0021.Module_1_FSoE.FSoE_Outputs.FSOE/FSOUT_Module_4_Channel_1_Output_X7_5 <-> Module 1 (FSoE)/FSoE Outputs/FSOE/FSOUT Module 4.Channel 1.Output (X7.5)
//     PlcTask Outputs/GVL_iXlinker.EtherCAT_Master_EKxxxx.Beckhoff_EKx9xx.Beckhoff_EKx9xxEK1122.A_0002_EK1960_0000_0021.Module_1_FSoE.FSoE_Outputs.FSOE/FSOUT_Module_4_Channel_2_Output_X7_6 <-> Module 1 (FSoE)/FSoE Outputs/FSOE/FSOUT Module 4.Channel 2.Output (X7.6)
//     PlcTask Outputs/GVL_iXlinker.EtherCAT_Master_EKxxxx.Beckhoff_EKx9xx.Beckhoff_EKx9xxEK1122.A_0002_EK1960_0000_0021.Module_1_FSoE.FSoE_Outputs.FSOE/FSOUT_Module_4_Channel_3_Output_X7_7 <-> Module 1 (FSoE)/FSoE Outputs/FSOE/FSOUT Module 4.Channel 3.Output (X7.7)
//     PlcTask Outputs/GVL_iXlinker.EtherCAT_Master_EKxxxx.Beckhoff_EKx9xx.Beckhoff_EKx9xxEK1122.A_0002_EK1960_0000_0021.Module_1_FSoE.FSoE_Outputs.FSOE/FSOUT_Module_4_Channel_4_Output_X7_8 <-> Module 1 (FSoE)/FSoE Outputs/FSOE/FSOUT Module 4.Channel 4.Output (X7.8)
//     PlcTask Outputs/GVL_iXlinker.EtherCAT_Master_EKxxxx.Beckhoff_EKx9xx.Beckhoff_EKx9xxEK1122.A_0002_EK1960_0000_0021.Module_1_FSoE.FSoE_Outputs.FSOE/FSOUT_Module_5_Channel_1_Output_X9_1 <-> Module 1 (FSoE)/FSoE Outputs/FSOE/FSOUT Module 5.Channel 1.Output (X9.1)
//     PlcTask Outputs/GVL_iXlinker.EtherCAT_Master_EKxxxx.Beckhoff_EKx9xx.Beckhoff_EKx9xxEK1122.A_0002_EK1960_0000_0021.Module_1_FSoE.FSoE_Outputs.FSOE/FSOUT_Module_5_Channel_2_Output_X9_2 <-> Module 1 (FSoE)/FSoE Outputs/FSOE/FSOUT Module 5.Channel 2.Output (X9.2)
//     PlcTask Outputs/GVL_iXlinker.EtherCAT_Master_EKxxxx.Beckhoff_EKx9xx.Beckhoff_EKx9xxEK1122.A_0002_EK1960_0000_0021.Module_1_FSoE.FSoE_Outputs.FSOE/FSOUT_Module_5_Channel_3_Output_X9_3 <-> Module 1 (FSoE)/FSoE Outputs/FSOE/FSOUT Module 5.Channel 3.Output (X9.3)
//     PlcTask Outputs/GVL_iXlinker.EtherCAT_Master_EKxxxx.Beckhoff_EKx9xx.Beckhoff_EKx9xxEK1122.A_0002_EK1960_0000_0021.Module_1_FSoE.FSoE_Outputs.FSOE/FSOUT_Module_5_Channel_4_Output_X9_4 <-> Module 1 (FSoE)/FSoE Outputs/FSOE/FSOUT Module 5.Channel 4.Output (X9.4)
//     PlcTask Outputs/GVL_iXlinker.EtherCAT_Master_EKxxxx.Beckhoff_EKx9xx.Beckhoff_EKx9xxEK1122.A_0002_EK1960_0000_0021.Module_1_FSoE.FSoE_Outputs.FSOE/FSOUT_Module_6_Channel_1_Output_X9_5 <-> Module 1 (FSoE)/FSoE Outputs/FSOE/FSOUT Module 6.Channel 1.Output (X9.5)
//     PlcTask Outputs/GVL_iXlinker.EtherCAT_Master_EKxxxx.Beckhoff_EKx9xx.Beckhoff_EKx9xxEK1122.A_0002_EK1960_0000_0021.Module_1_FSoE.FSoE_Outputs.FSOE/FSOUT_Module_6_Channel_2_Output_X9_6 <-> Module 1 (FSoE)/FSoE Outputs/FSOE/FSOUT Module 6.Channel 2.Output (X9.6)
//     PlcTask Outputs/GVL_iXlinker.EtherCAT_Master_EKxxxx.Beckhoff_EKx9xx.Beckhoff_EKx9xxEK1122.A_0002_EK1960_0000_0021.Module_1_FSoE.FSoE_Outputs.FSOE/FSOUT_Module_6_Channel_3_Output_X9_7 <-> Module 1 (FSoE)/FSoE Outputs/FSOE/FSOUT Module 6.Channel 3.Output (X9.7)
//     PlcTask Outputs/GVL_iXlinker.EtherCAT_Master_EKxxxx.Beckhoff_EKx9xx.Beckhoff_EKx9xxEK1122.A_0002_EK1960_0000_0021.Module_1_FSoE.FSoE_Outputs.FSOE/FSOUT_Module_6_Channel_4_Output_X9_8 <-> Module 1 (FSoE)/FSoE Outputs/FSOE/FSOUT Module 6.Channel 4.Output (X9.8)
//     PlcTask Outputs/GVL_iXlinker.EtherCAT_Master_EKxxxx.Beckhoff_EKx9xx.Beckhoff_EKx9xxEK1122.A_0002_EK1960_0000_0021.Module_1_FSoE.FSoE_Outputs.FSOE/FSOUT_Module_1_ErrAck <-> Module 1 (FSoE)/FSoE Outputs/FSOE/FSOUT Module 1.ErrAck
//     PlcTask Outputs/GVL_iXlinker.EtherCAT_Master_EKxxxx.Beckhoff_EKx9xx.Beckhoff_EKx9xxEK1122.A_0002_EK1960_0000_0021.Module_1_FSoE.FSoE_Outputs.FSOE/FSOUT_Module_2_ErrAck <-> Module 1 (FSoE)/FSoE Outputs/FSOE/FSOUT Module 2.ErrAck
//     PlcTask Outputs/GVL_iXlinker.EtherCAT_Master_EKxxxx.Beckhoff_EKx9xx.Beckhoff_EKx9xxEK1122.A_0002_EK1960_0000_0021.Module_1_FSoE.FSoE_Outputs.FSOE/FSOUT_Module_3_ErrAck <-> Module 1 (FSoE)/FSoE Outputs/FSOE/FSOUT Module 3.ErrAck
//     PlcTask Outputs/GVL_iXlinker.EtherCAT_Master_EKxxxx.Beckhoff_EKx9xx.Beckhoff_EKx9xxEK1122.A_0002_EK1960_0000_0021.Module_1_FSoE.FSoE_Outputs.FSOE/FSOUT_Module_4_ErrAck <-> Module 1 (FSoE)/FSoE Outputs/FSOE/FSOUT Module 4.ErrAck
//     PlcTask Outputs/GVL_iXlinker.EtherCAT_Master_EKxxxx.Beckhoff_EKx9xx.Beckhoff_EKx9xxEK1122.A_0002_EK1960_0000_0021.Module_1_FSoE.FSoE_Outputs.FSOE/FSOUT_Module_5_ErrAck <-> Module 1 (FSoE)/FSoE Outputs/FSOE/FSOUT Module 5.ErrAck
//     PlcTask Outputs/GVL_iXlinker.EtherCAT_Master_EKxxxx.Beckhoff_EKx9xx.Beckhoff_EKx9xxEK1122.A_0002_EK1960_0000_0021.Module_1_FSoE.FSoE_Outputs.FSOE/FSOUT_Module_6_ErrAck <-> Module 1 (FSoE)/FSoE Outputs/FSOE/FSOUT Module 6.ErrAck
//     PlcTask Outputs/GVL_iXlinker.EtherCAT_Master_EKxxxx.Beckhoff_EKx9xx.Beckhoff_EKx9xxEK1122.A_0002_EK1960_0000_0021.Module_1_FSoE.FSoE_Outputs.FSOE/FSoE_CRC_000 <-> Module 1 (FSoE)/FSoE Outputs/FSOE/FSoE CRC 000
//     PlcTask Outputs/GVL_iXlinker.EtherCAT_Master_EKxxxx.Beckhoff_EKx9xx.Beckhoff_EKx9xxEK1122.A_0002_EK1960_0000_0021.Module_1_FSoE.FSoE_Outputs.FSOE/FSoE_CRC_001 <-> Module 1 (FSoE)/FSoE Outputs/FSOE/FSoE CRC 001
//     PlcTask Outputs/GVL_iXlinker.EtherCAT_Master_EKxxxx.Beckhoff_EKx9xx.Beckhoff_EKx9xxEK1122.A_0002_EK1960_0000_0021.Module_1_FSoE.FSoE_Outputs.FSOE/FSoE_CRC_002 <-> Module 1 (FSoE)/FSoE Outputs/FSOE/FSoE CRC 002
//     PlcTask Outputs/GVL_iXlinker.EtherCAT_Master_EKxxxx.Beckhoff_EKx9xx.Beckhoff_EKx9xxEK1122.A_0002_EK1960_0000_0021.Module_1_FSoE.FSoE_Outputs.FSOE/FSIN_Module_1_ErrAck <-> Module 1 (FSoE)/FSoE Outputs/FSOE/FSIN Module 1.ErrAck
//     PlcTask Outputs/GVL_iXlinker.EtherCAT_Master_EKxxxx.Beckhoff_EKx9xx.Beckhoff_EKx9xxEK1122.A_0002_EK1960_0000_0021.Module_1_FSoE.FSoE_Outputs.FSOE/FSIN_Module_2_ErrAck <-> Module 1 (FSoE)/FSoE Outputs/FSOE/FSIN Module 2.ErrAck
//     PlcTask Outputs/GVL_iXlinker.EtherCAT_Master_EKxxxx.Beckhoff_EKx9xx.Beckhoff_EKx9xxEK1122.A_0002_EK1960_0000_0021.Module_1_FSoE.FSoE_Outputs.FSOE/FSIN_Module_3_ErrAck <-> Module 1 (FSoE)/FSoE Outputs/FSOE/FSIN Module 3.ErrAck
//     PlcTask Outputs/GVL_iXlinker.EtherCAT_Master_EKxxxx.Beckhoff_EKx9xx.Beckhoff_EKx9xxEK1122.A_0002_EK1960_0000_0021.Module_1_FSoE.FSoE_Outputs.FSOE/FSIN_Module_4_ErrAck <-> Module 1 (FSoE)/FSoE Outputs/FSOE/FSIN Module 4.ErrAck
//     PlcTask Outputs/GVL_iXlinker.EtherCAT_Master_EKxxxx.Beckhoff_EKx9xx.Beckhoff_EKx9xxEK1122.A_0002_EK1960_0000_0021.Module_1_FSoE.FSoE_Outputs.FSOE/FSIN_Module_5_ErrAck <-> Module 1 (FSoE)/FSoE Outputs/FSOE/FSIN Module 5.ErrAck
//     PlcTask Outputs/GVL_iXlinker.EtherCAT_Master_EKxxxx.Beckhoff_EKx9xx.Beckhoff_EKx9xxEK1122.A_0002_EK1960_0000_0021.Module_1_FSoE.FSoE_Outputs.FSOE/FSIN_Module_6_ErrAck <-> Module 1 (FSoE)/FSoE Outputs/FSOE/FSIN Module 6.ErrAck
//     PlcTask Outputs/GVL_iXlinker.EtherCAT_Master_EKxxxx.Beckhoff_EKx9xx.Beckhoff_EKx9xxEK1122.A_0002_EK1960_0000_0021.Module_1_FSoE.FSoE_Outputs.FSOE/FSIN_Module_7_ErrAck <-> Module 1 (FSoE)/FSoE Outputs/FSOE/FSIN Module 7.ErrAck
//     PlcTask Outputs/GVL_iXlinker.EtherCAT_Master_EKxxxx.Beckhoff_EKx9xx.Beckhoff_EKx9xxEK1122.A_0002_EK1960_0000_0021.Module_1_FSoE.FSoE_Outputs.FSOE/FSIN_Module_8_ErrAck <-> Module 1 (FSoE)/FSoE Outputs/FSOE/FSIN Module 8.ErrAck
//     PlcTask Outputs/GVL_iXlinker.EtherCAT_Master_EKxxxx.Beckhoff_EKx9xx.Beckhoff_EKx9xxEK1122.A_0002_EK1960_0000_0021.Module_1_FSoE.FSoE_Outputs.FSOE/FSIN_Module_9_Err_Ack_1 <-> Module 1 (FSoE)/FSoE Outputs/FSOE/FSIN Module 9.Err Ack 1
//     PlcTask Outputs/GVL_iXlinker.EtherCAT_Master_EKxxxx.Beckhoff_EKx9xx.Beckhoff_EKx9xxEK1122.A_0002_EK1960_0000_0021.Module_1_FSoE.FSoE_Outputs.FSOE/FSIN_Module_9_Err_Ack_2 <-> Module 1 (FSoE)/FSoE Outputs/FSOE/FSIN Module 9.Err Ack 2
//     PlcTask Outputs/GVL_iXlinker.EtherCAT_Master_EKxxxx.Beckhoff_EKx9xx.Beckhoff_EKx9xxEK1122.A_0002_EK1960_0000_0021.Module_1_FSoE.FSoE_Outputs.FSOE/FSIN_Module_10_Err_Ack_1 <-> Module 1 (FSoE)/FSoE Outputs/FSOE/FSIN Module 10.Err Ack 1
//     PlcTask Outputs/GVL_iXlinker.EtherCAT_Master_EKxxxx.Beckhoff_EKx9xx.Beckhoff_EKx9xxEK1122.A_0002_EK1960_0000_0021.Module_1_FSoE.FSoE_Outputs.FSOE/FSIN_Module_10_Err_Ack_2 <-> Module 1 (FSoE)/FSoE Outputs/FSOE/FSIN Module 10.Err Ack 2
//     PlcTask Outputs/GVL_iXlinker.EtherCAT_Master_EKxxxx.Beckhoff_EKx9xx.Beckhoff_EKx9xxEK1122.A_0002_EK1960_0000_0021.Module_1_FSoE.FSoE_Outputs.FSOE/FSoE_Connection_ID <-> Module 1 (FSoE)/FSoE Outputs/FSOE/FSoE Connection ID
//     PlcTask Outputs/GVL_iXlinker.EtherCAT_Master_EKxxxx.Beckhoff_EKx9xx.Beckhoff_EKx9xxEK1122.A_0002_EK1960_0000_0021.Module_2_FSOUT.Outputs.Module_1_Channel_1_Standard_Output_X5_1 <-> Module 2 (FSOUT)/Outputs/Module 1.Channel 1.Standard Output (X5.1)
//     PlcTask Outputs/GVL_iXlinker.EtherCAT_Master_EKxxxx.Beckhoff_EKx9xx.Beckhoff_EKx9xxEK1122.A_0002_EK1960_0000_0021.Module_2_FSOUT.Outputs.Module_1_Channel_2_Standard_Output_X5_2 <-> Module 2 (FSOUT)/Outputs/Module 1.Channel 2.Standard Output (X5.2)
//     PlcTask Outputs/GVL_iXlinker.EtherCAT_Master_EKxxxx.Beckhoff_EKx9xx.Beckhoff_EKx9xxEK1122.A_0002_EK1960_0000_0021.Module_2_FSOUT.Outputs.Module_1_Channel_3_Standard_Output_X5_3 <-> Module 2 (FSOUT)/Outputs/Module 1.Channel 3.Standard Output (X5.3)
//     PlcTask Outputs/GVL_iXlinker.EtherCAT_Master_EKxxxx.Beckhoff_EKx9xx.Beckhoff_EKx9xxEK1122.A_0002_EK1960_0000_0021.Module_2_FSOUT.Outputs.Module_1_Channel_4_Standard_Output_X5_4 <-> Module 2 (FSOUT)/Outputs/Module 1.Channel 4.Standard Output (X5.4)
//     PlcTask Outputs/GVL_iXlinker.EtherCAT_Master_EKxxxx.Beckhoff_EKx9xx.Beckhoff_EKx9xxEK1122.A_0002_EK1960_0000_0021.Module_2_FSOUT.Outputs.Module_2_Channel_1_Standard_Output_X5_5 <-> Module 2 (FSOUT)/Outputs/Module 2.Channel 1.Standard Output (X5.5)
//     PlcTask Outputs/GVL_iXlinker.EtherCAT_Master_EKxxxx.Beckhoff_EKx9xx.Beckhoff_EKx9xxEK1122.A_0002_EK1960_0000_0021.Module_2_FSOUT.Outputs.Module_2_Channel_2_Standard_Output_X5_6 <-> Module 2 (FSOUT)/Outputs/Module 2.Channel 2.Standard Output (X5.6)
//     PlcTask Outputs/GVL_iXlinker.EtherCAT_Master_EKxxxx.Beckhoff_EKx9xx.Beckhoff_EKx9xxEK1122.A_0002_EK1960_0000_0021.Module_2_FSOUT.Outputs.Module_2_Channel_3_Standard_Output_X5_7 <-> Module 2 (FSOUT)/Outputs/Module 2.Channel 3.Standard Output (X5.7)
//     PlcTask Outputs/GVL_iXlinker.EtherCAT_Master_EKxxxx.Beckhoff_EKx9xx.Beckhoff_EKx9xxEK1122.A_0002_EK1960_0000_0021.Module_2_FSOUT.Outputs.Module_2_Channel_4_Standard_Output_X5_8 <-> Module 2 (FSOUT)/Outputs/Module 2.Channel 4.Standard Output (X5.8)
//     PlcTask Outputs/GVL_iXlinker.EtherCAT_Master_EKxxxx.Beckhoff_EKx9xx.Beckhoff_EKx9xxEK1122.A_0002_EK1960_0000_0021.Module_2_FSOUT.Outputs.Module_3_Channel_1_Standard_Output_X7_1 <-> Module 2 (FSOUT)/Outputs/Module 3.Channel 1.Standard Output (X7.1)
//     PlcTask Outputs/GVL_iXlinker.EtherCAT_Master_EKxxxx.Beckhoff_EKx9xx.Beckhoff_EKx9xxEK1122.A_0002_EK1960_0000_0021.Module_2_FSOUT.Outputs.Module_3_Channel_2_Standard_Output_X7_2 <-> Module 2 (FSOUT)/Outputs/Module 3.Channel 2.Standard Output (X7.2)
//     PlcTask Outputs/GVL_iXlinker.EtherCAT_Master_EKxxxx.Beckhoff_EKx9xx.Beckhoff_EKx9xxEK1122.A_0002_EK1960_0000_0021.Module_2_FSOUT.Outputs.Module_3_Channel_3_Standard_Output_X7_3 <-> Module 2 (FSOUT)/Outputs/Module 3.Channel 3.Standard Output (X7.3)
//     PlcTask Outputs/GVL_iXlinker.EtherCAT_Master_EKxxxx.Beckhoff_EKx9xx.Beckhoff_EKx9xxEK1122.A_0002_EK1960_0000_0021.Module_2_FSOUT.Outputs.Module_3_Channel_4_Standard_Output_X7_4 <-> Module 2 (FSOUT)/Outputs/Module 3.Channel 4.Standard Output (X7.4)
//     PlcTask Outputs/GVL_iXlinker.EtherCAT_Master_EKxxxx.Beckhoff_EKx9xx.Beckhoff_EKx9xxEK1122.A_0002_EK1960_0000_0021.Module_2_FSOUT.Outputs.Module_4_Channel_1_Standard_Output_X7_5 <-> Module 2 (FSOUT)/Outputs/Module 4.Channel 1.Standard Output (X7.5)
//     PlcTask Outputs/GVL_iXlinker.EtherCAT_Master_EKxxxx.Beckhoff_EKx9xx.Beckhoff_EKx9xxEK1122.A_0002_EK1960_0000_0021.Module_2_FSOUT.Outputs.Module_4_Channel_2_Standard_Output_X7_6 <-> Module 2 (FSOUT)/Outputs/Module 4.Channel 2.Standard Output (X7.6)
//     PlcTask Outputs/GVL_iXlinker.EtherCAT_Master_EKxxxx.Beckhoff_EKx9xx.Beckhoff_EKx9xxEK1122.A_0002_EK1960_0000_0021.Module_2_FSOUT.Outputs.Module_4_Channel_3_Standard_Output_X7_7 <-> Module 2 (FSOUT)/Outputs/Module 4.Channel 3.Standard Output (X7.7)
//     PlcTask Outputs/GVL_iXlinker.EtherCAT_Master_EKxxxx.Beckhoff_EKx9xx.Beckhoff_EKx9xxEK1122.A_0002_EK1960_0000_0021.Module_2_FSOUT.Outputs.Module_4_Channel_4_Standard_Output_X7_8 <-> Module 2 (FSOUT)/Outputs/Module 4.Channel 4.Standard Output (X7.8)
//     PlcTask Outputs/GVL_iXlinker.EtherCAT_Master_EKxxxx.Beckhoff_EKx9xx.Beckhoff_EKx9xxEK1122.A_0002_EK1960_0000_0021.Module_2_FSOUT.Outputs.Module_5_Channel_1_Standard_Output_X9_1 <-> Module 2 (FSOUT)/Outputs/Module 5.Channel 1.Standard Output (X9.1)
//     PlcTask Outputs/GVL_iXlinker.EtherCAT_Master_EKxxxx.Beckhoff_EKx9xx.Beckhoff_EKx9xxEK1122.A_0002_EK1960_0000_0021.Module_2_FSOUT.Outputs.Module_5_Channel_2_Standard_Output_X9_2 <-> Module 2 (FSOUT)/Outputs/Module 5.Channel 2.Standard Output (X9.2)
//     PlcTask Outputs/GVL_iXlinker.EtherCAT_Master_EKxxxx.Beckhoff_EKx9xx.Beckhoff_EKx9xxEK1122.A_0002_EK1960_0000_0021.Module_2_FSOUT.Outputs.Module_5_Channel_3_Standard_Output_X9_3 <-> Module 2 (FSOUT)/Outputs/Module 5.Channel 3.Standard Output (X9.3)
//     PlcTask Outputs/GVL_iXlinker.EtherCAT_Master_EKxxxx.Beckhoff_EKx9xx.Beckhoff_EKx9xxEK1122.A_0002_EK1960_0000_0021.Module_2_FSOUT.Outputs.Module_5_Channel_4_Standard_Output_X9_4 <-> Module 2 (FSOUT)/Outputs/Module 5.Channel 4.Standard Output (X9.4)
//     PlcTask Outputs/GVL_iXlinker.EtherCAT_Master_EKxxxx.Beckhoff_EKx9xx.Beckhoff_EKx9xxEK1122.A_0002_EK1960_0000_0021.Module_2_FSOUT.Outputs.Module_6_Channel_1_Standard_Output_X9_5 <-> Module 2 (FSOUT)/Outputs/Module 6.Channel 1.Standard Output (X9.5)
//     PlcTask Outputs/GVL_iXlinker.EtherCAT_Master_EKxxxx.Beckhoff_EKx9xx.Beckhoff_EKx9xxEK1122.A_0002_EK1960_0000_0021.Module_2_FSOUT.Outputs.Module_6_Channel_2_Standard_Output_X9_6 <-> Module 2 (FSOUT)/Outputs/Module 6.Channel 2.Standard Output (X9.6)
//     PlcTask Outputs/GVL_iXlinker.EtherCAT_Master_EKxxxx.Beckhoff_EKx9xx.Beckhoff_EKx9xxEK1122.A_0002_EK1960_0000_0021.Module_2_FSOUT.Outputs.Module_6_Channel_3_Standard_Output_X9_7 <-> Module 2 (FSOUT)/Outputs/Module 6.Channel 3.Standard Output (X9.7)
//     PlcTask Outputs/GVL_iXlinker.EtherCAT_Master_EKxxxx.Beckhoff_EKx9xx.Beckhoff_EKx9xxEK1122.A_0002_EK1960_0000_0021.Module_2_FSOUT.Outputs.Module_6_Channel_4_Standard_Output_X9_8 <-> Module 2 (FSOUT)/Outputs/Module 6.Channel 4.Standard Output (X9.8)
//     PlcTask Inputs/GVL_iXlinker.EtherCAT_Master_EKxxxx.Beckhoff_EKx9xx.Beckhoff_EKx9xxEK1122.A_0002_EK1960_0000_0021.Module_3_FSLOGIC.FSLOGIC_Inputs.Safe_Logic_State <-> Module 3 (FSLOGIC)/FSLOGIC Inputs/Safe Logic State
//     PlcTask Inputs/GVL_iXlinker.EtherCAT_Master_EKxxxx.Beckhoff_EKx9xx.Beckhoff_EKx9xxEK1122.A_0002_EK1960_0000_0021.Module_3_FSLOGIC.FSLOGIC_Inputs.Cycle_Counter <-> Module 3 (FSLOGIC)/FSLOGIC Inputs/Cycle Counter
//     PlcTask Inputs/GVL_iXlinker.EtherCAT_Master_EKxxxx.Beckhoff_EKx9xx.Beckhoff_EKx9xxEK1122.A_0002_EK1960_0000_0021.WcState.WcState0 <-> WcState/WcState0
//     PlcTask Inputs/GVL_iXlinker.EtherCAT_Master_EKxxxx.Beckhoff_EKx9xx.Beckhoff_EKx9xxEK1122.A_0002_EK1960_0000_0021.WcState.WcState1 <-> WcState/WcState1
//     PlcTask Inputs/GVL_iXlinker.EtherCAT_Master_EKxxxx.Beckhoff_EKx9xx.Beckhoff_EKx9xxEK1122.A_0002_EK1960_0000_0021.WcState.InputToggle0 <-> WcState/InputToggle0
//     PlcTask Inputs/GVL_iXlinker.EtherCAT_Master_EKxxxx.Beckhoff_EKx9xx.Beckhoff_EKx9xxEK1122.A_0002_EK1960_0000_0021.WcState.InputToggle1 <-> WcState/InputToggle1
//     PlcTask Inputs/GVL_iXlinker.EtherCAT_Master_EKxxxx.Beckhoff_EKx9xx.Beckhoff_EKx9xxEK1122.A_0002_EK1960_0000_0021.InfoData.AdsAddr <-> InfoData/AdsAddr
//     PlcTask Inputs/GVL_iXlinker.EtherCAT_Master_EKxxxx.Beckhoff_EKx9xx.Beckhoff_EKx9xxEK1122.A_0002_EK1960_0000_0021.InfoData.State <-> InfoData/State
//   PLC/PLC Instance <-> EtherCAT Master EKxxxx/Beckhoff EKx9xx/Beckhoff EKx9xxEK1122/A_0003(EK1960-0008-0019)
//     PlcTask Inputs/GVL_iXlinker.EtherCAT_Master_EKxxxx.Beckhoff_EKx9xx.Beckhoff_EKx9xxEK1122.A_0003_EK1960_0008_0019.Module_1_FSoE.FSoE_Inputs.FSOE/FSoE_Command <-> Module 1 (FSoE)/FSoE Inputs/FSOE/FSoE Command
//     PlcTask Inputs/GVL_iXlinker.EtherCAT_Master_EKxxxx.Beckhoff_EKx9xx.Beckhoff_EKx9xxEK1122.A_0003_EK1960_0008_0019.Module_1_FSoE.FSoE_Inputs.FSOE/FSOUT_Module_1_Module_Fault <-> Module 1 (FSoE)/FSoE Inputs/FSOE/FSOUT Module 1.Module Fault
//     PlcTask Inputs/GVL_iXlinker.EtherCAT_Master_EKxxxx.Beckhoff_EKx9xx.Beckhoff_EKx9xxEK1122.A_0003_EK1960_0008_0019.Module_1_FSoE.FSoE_Inputs.FSOE/FSOUT_Module_2_Module_Fault <-> Module 1 (FSoE)/FSoE Inputs/FSOE/FSOUT Module 2.Module Fault
//     PlcTask Inputs/GVL_iXlinker.EtherCAT_Master_EKxxxx.Beckhoff_EKx9xx.Beckhoff_EKx9xxEK1122.A_0003_EK1960_0008_0019.Module_1_FSoE.FSoE_Inputs.FSOE/FSOUT_Module_3_Module_Fault <-> Module 1 (FSoE)/FSoE Inputs/FSOE/FSOUT Module 3.Module Fault
//     PlcTask Inputs/GVL_iXlinker.EtherCAT_Master_EKxxxx.Beckhoff_EKx9xx.Beckhoff_EKx9xxEK1122.A_0003_EK1960_0008_0019.Module_1_FSoE.FSoE_Inputs.FSOE/FSOUT_Module_4_Module_Fault <-> Module 1 (FSoE)/FSoE Inputs/FSOE/FSOUT Module 4.Module Fault
//     PlcTask Inputs/GVL_iXlinker.EtherCAT_Master_EKxxxx.Beckhoff_EKx9xx.Beckhoff_EKx9xxEK1122.A_0003_EK1960_0008_0019.Module_1_FSoE.FSoE_Inputs.FSOE/FSOUT_Module_5_Module_Fault <-> Module 1 (FSoE)/FSoE Inputs/FSOE/FSOUT Module 5.Module Fault
//     PlcTask Inputs/GVL_iXlinker.EtherCAT_Master_EKxxxx.Beckhoff_EKx9xx.Beckhoff_EKx9xxEK1122.A_0003_EK1960_0008_0019.Module_1_FSoE.FSoE_Inputs.FSOE/FSOUT_Module_6_Module_Fault <-> Module 1 (FSoE)/FSoE Inputs/FSOE/FSOUT Module 6.Module Fault
//     PlcTask Inputs/GVL_iXlinker.EtherCAT_Master_EKxxxx.Beckhoff_EKx9xx.Beckhoff_EKx9xxEK1122.A_0003_EK1960_0008_0019.Module_1_FSoE.FSoE_Inputs.FSOE/FSIN_Module_1_Channel_1_Input <-> Module 1 (FSoE)/FSoE Inputs/FSOE/FSIN Module 1.Channel 1.Input
//     PlcTask Inputs/GVL_iXlinker.EtherCAT_Master_EKxxxx.Beckhoff_EKx9xx.Beckhoff_EKx9xxEK1122.A_0003_EK1960_0008_0019.Module_1_FSoE.FSoE_Inputs.FSOE/FSIN_Module_1_Channel_2_Input <-> Module 1 (FSoE)/FSoE Inputs/FSOE/FSIN Module 1.Channel 2.Input
//     PlcTask Inputs/GVL_iXlinker.EtherCAT_Master_EKxxxx.Beckhoff_EKx9xx.Beckhoff_EKx9xxEK1122.A_0003_EK1960_0008_0019.Module_1_FSoE.FSoE_Inputs.FSOE/FSIN_Module_2_Channel_1_Input <-> Module 1 (FSoE)/FSoE Inputs/FSOE/FSIN Module 2.Channel 1.Input
//     PlcTask Inputs/GVL_iXlinker.EtherCAT_Master_EKxxxx.Beckhoff_EKx9xx.Beckhoff_EKx9xxEK1122.A_0003_EK1960_0008_0019.Module_1_FSoE.FSoE_Inputs.FSOE/FSIN_Module_2_Channel_2_Input <-> Module 1 (FSoE)/FSoE Inputs/FSOE/FSIN Module 2.Channel 2.Input
//     PlcTask Inputs/GVL_iXlinker.EtherCAT_Master_EKxxxx.Beckhoff_EKx9xx.Beckhoff_EKx9xxEK1122.A_0003_EK1960_0008_0019.Module_1_FSoE.FSoE_Inputs.FSOE/FSIN_Module_3_Channel_1_Input <-> Module 1 (FSoE)/FSoE Inputs/FSOE/FSIN Module 3.Channel 1.Input
//     PlcTask Inputs/GVL_iXlinker.EtherCAT_Master_EKxxxx.Beckhoff_EKx9xx.Beckhoff_EKx9xxEK1122.A_0003_EK1960_0008_0019.Module_1_FSoE.FSoE_Inputs.FSOE/FSIN_Module_3_Channel_2_Input <-> Module 1 (FSoE)/FSoE Inputs/FSOE/FSIN Module 3.Channel 2.Input
//     PlcTask Inputs/GVL_iXlinker.EtherCAT_Master_EKxxxx.Beckhoff_EKx9xx.Beckhoff_EKx9xxEK1122.A_0003_EK1960_0008_0019.Module_1_FSoE.FSoE_Inputs.FSOE/FSIN_Module_4_Channel_1_Input <-> Module 1 (FSoE)/FSoE Inputs/FSOE/FSIN Module 4.Channel 1.Input
//     PlcTask Inputs/GVL_iXlinker.EtherCAT_Master_EKxxxx.Beckhoff_EKx9xx.Beckhoff_EKx9xxEK1122.A_0003_EK1960_0008_0019.Module_1_FSoE.FSoE_Inputs.FSOE/FSIN_Module_4_Channel_2_Input <-> Module 1 (FSoE)/FSoE Inputs/FSOE/FSIN Module 4.Channel 2.Input
//     PlcTask Inputs/GVL_iXlinker.EtherCAT_Master_EKxxxx.Beckhoff_EKx9xx.Beckhoff_EKx9xxEK1122.A_0003_EK1960_0008_0019.Module_1_FSoE.FSoE_Inputs.FSOE/FSIN_Module_5_Channel_1_Input <-> Module 1 (FSoE)/FSoE Inputs/FSOE/FSIN Module 5.Channel 1.Input
//     PlcTask Inputs/GVL_iXlinker.EtherCAT_Master_EKxxxx.Beckhoff_EKx9xx.Beckhoff_EKx9xxEK1122.A_0003_EK1960_0008_0019.Module_1_FSoE.FSoE_Inputs.FSOE/FSIN_Module_5_Channel_2_Input <-> Module 1 (FSoE)/FSoE Inputs/FSOE/FSIN Module 5.Channel 2.Input
//     PlcTask Inputs/GVL_iXlinker.EtherCAT_Master_EKxxxx.Beckhoff_EKx9xx.Beckhoff_EKx9xxEK1122.A_0003_EK1960_0008_0019.Module_1_FSoE.FSoE_Inputs.FSOE/FSIN_Module_6_Channel_1_Input <-> Module 1 (FSoE)/FSoE Inputs/FSOE/FSIN Module 6.Channel 1.Input
//     PlcTask Inputs/GVL_iXlinker.EtherCAT_Master_EKxxxx.Beckhoff_EKx9xx.Beckhoff_EKx9xxEK1122.A_0003_EK1960_0008_0019.Module_1_FSoE.FSoE_Inputs.FSOE/FSIN_Module_6_Channel_2_Input <-> Module 1 (FSoE)/FSoE Inputs/FSOE/FSIN Module 6.Channel 2.Input
//     PlcTask Inputs/GVL_iXlinker.EtherCAT_Master_EKxxxx.Beckhoff_EKx9xx.Beckhoff_EKx9xxEK1122.A_0003_EK1960_0008_0019.Module_1_FSoE.FSoE_Inputs.FSOE/FSIN_Module_7_Channel_1_Input <-> Module 1 (FSoE)/FSoE Inputs/FSOE/FSIN Module 7.Channel 1.Input
//     PlcTask Inputs/GVL_iXlinker.EtherCAT_Master_EKxxxx.Beckhoff_EKx9xx.Beckhoff_EKx9xxEK1122.A_0003_EK1960_0008_0019.Module_1_FSoE.FSoE_Inputs.FSOE/FSIN_Module_7_Channel_2_Input <-> Module 1 (FSoE)/FSoE Inputs/FSOE/FSIN Module 7.Channel 2.Input
//     PlcTask Inputs/GVL_iXlinker.EtherCAT_Master_EKxxxx.Beckhoff_EKx9xx.Beckhoff_EKx9xxEK1122.A_0003_EK1960_0008_0019.Module_1_FSoE.FSoE_Inputs.FSOE/FSIN_Module_8_Channel_1_Input <-> Module 1 (FSoE)/FSoE Inputs/FSOE/FSIN Module 8.Channel 1.Input
//     PlcTask Inputs/GVL_iXlinker.EtherCAT_Master_EKxxxx.Beckhoff_EKx9xx.Beckhoff_EKx9xxEK1122.A_0003_EK1960_0008_0019.Module_1_FSoE.FSoE_Inputs.FSOE/FSIN_Module_8_Channel_2_Input <-> Module 1 (FSoE)/FSoE Inputs/FSOE/FSIN Module 8.Channel 2.Input
//     PlcTask Inputs/GVL_iXlinker.EtherCAT_Master_EKxxxx.Beckhoff_EKx9xx.Beckhoff_EKx9xxEK1122.A_0003_EK1960_0008_0019.Module_1_FSoE.FSoE_Inputs.FSOE/FSIN_Module_9_Channel_1_Input <-> Module 1 (FSoE)/FSoE Inputs/FSOE/FSIN Module 9.Channel 1.Input
//     PlcTask Inputs/GVL_iXlinker.EtherCAT_Master_EKxxxx.Beckhoff_EKx9xx.Beckhoff_EKx9xxEK1122.A_0003_EK1960_0008_0019.Module_1_FSoE.FSoE_Inputs.FSOE/FSIN_Module_9_Channel_2_Input <-> Module 1 (FSoE)/FSoE Inputs/FSOE/FSIN Module 9.Channel 2.Input
//     PlcTask Inputs/GVL_iXlinker.EtherCAT_Master_EKxxxx.Beckhoff_EKx9xx.Beckhoff_EKx9xxEK1122.A_0003_EK1960_0008_0019.Module_1_FSoE.FSoE_Inputs.FSOE/FSIN_Module_10_Channel_1_Input <-> Module 1 (FSoE)/FSoE Inputs/FSOE/FSIN Module 10.Channel 1.Input
//     PlcTask Inputs/GVL_iXlinker.EtherCAT_Master_EKxxxx.Beckhoff_EKx9xx.Beckhoff_EKx9xxEK1122.A_0003_EK1960_0008_0019.Module_1_FSoE.FSoE_Inputs.FSOE/FSIN_Module_10_Channel_2_Input <-> Module 1 (FSoE)/FSoE Inputs/FSOE/FSIN Module 10.Channel 2.Input
//     PlcTask Inputs/GVL_iXlinker.EtherCAT_Master_EKxxxx.Beckhoff_EKx9xx.Beckhoff_EKx9xxEK1122.A_0003_EK1960_0008_0019.Module_1_FSoE.FSoE_Inputs.FSOE/FSIN_Module_1_Module_Fault <-> Module 1 (FSoE)/FSoE Inputs/FSOE/FSIN Module 1.Module Fault
//     PlcTask Inputs/GVL_iXlinker.EtherCAT_Master_EKxxxx.Beckhoff_EKx9xx.Beckhoff_EKx9xxEK1122.A_0003_EK1960_0008_0019.Module_1_FSoE.FSoE_Inputs.FSOE/FSIN_Module_2_Module_Fault <-> Module 1 (FSoE)/FSoE Inputs/FSOE/FSIN Module 2.Module Fault
//     PlcTask Inputs/GVL_iXlinker.EtherCAT_Master_EKxxxx.Beckhoff_EKx9xx.Beckhoff_EKx9xxEK1122.A_0003_EK1960_0008_0019.Module_1_FSoE.FSoE_Inputs.FSOE/FSIN_Module_3_Module_Fault <-> Module 1 (FSoE)/FSoE Inputs/FSOE/FSIN Module 3.Module Fault
//     PlcTask Inputs/GVL_iXlinker.EtherCAT_Master_EKxxxx.Beckhoff_EKx9xx.Beckhoff_EKx9xxEK1122.A_0003_EK1960_0008_0019.Module_1_FSoE.FSoE_Inputs.FSOE/FSIN_Module_4_Module_Fault <-> Module 1 (FSoE)/FSoE Inputs/FSOE/FSIN Module 4.Module Fault
//     PlcTask Inputs/GVL_iXlinker.EtherCAT_Master_EKxxxx.Beckhoff_EKx9xx.Beckhoff_EKx9xxEK1122.A_0003_EK1960_0008_0019.Module_1_FSoE.FSoE_Inputs.FSOE/FSIN_Module_5_Module_Fault <-> Module 1 (FSoE)/FSoE Inputs/FSOE/FSIN Module 5.Module Fault
//     PlcTask Inputs/GVL_iXlinker.EtherCAT_Master_EKxxxx.Beckhoff_EKx9xx.Beckhoff_EKx9xxEK1122.A_0003_EK1960_0008_0019.Module_1_FSoE.FSoE_Inputs.FSOE/FSIN_Module_6_Module_Fault <-> Module 1 (FSoE)/FSoE Inputs/FSOE/FSIN Module 6.Module Fault
//     PlcTask Inputs/GVL_iXlinker.EtherCAT_Master_EKxxxx.Beckhoff_EKx9xx.Beckhoff_EKx9xxEK1122.A_0003_EK1960_0008_0019.Module_1_FSoE.FSoE_Inputs.FSOE/FSIN_Module_7_Module_Fault <-> Module 1 (FSoE)/FSoE Inputs/FSOE/FSIN Module 7.Module Fault
//     PlcTask Inputs/GVL_iXlinker.EtherCAT_Master_EKxxxx.Beckhoff_EKx9xx.Beckhoff_EKx9xxEK1122.A_0003_EK1960_0008_0019.Module_1_FSoE.FSoE_Inputs.FSOE/FSIN_Module_8_Module_Fault <-> Module 1 (FSoE)/FSoE Inputs/FSOE/FSIN Module 8.Module Fault
//     PlcTask Inputs/GVL_iXlinker.EtherCAT_Master_EKxxxx.Beckhoff_EKx9xx.Beckhoff_EKx9xxEK1122.A_0003_EK1960_0008_0019.Module_1_FSoE.FSoE_Inputs.FSOE/FSoE_CRC_000 <-> Module 1 (FSoE)/FSoE Inputs/FSOE/FSoE CRC 000
//     PlcTask Inputs/GVL_iXlinker.EtherCAT_Master_EKxxxx.Beckhoff_EKx9xx.Beckhoff_EKx9xxEK1122.A_0003_EK1960_0008_0019.Module_1_FSoE.FSoE_Inputs.FSOE/FSoE_CRC_001 <-> Module 1 (FSoE)/FSoE Inputs/FSOE/FSoE CRC 001
//     PlcTask Inputs/GVL_iXlinker.EtherCAT_Master_EKxxxx.Beckhoff_EKx9xx.Beckhoff_EKx9xxEK1122.A_0003_EK1960_0008_0019.Module_1_FSoE.FSoE_Inputs.FSOE/FSoE_CRC_002 <-> Module 1 (FSoE)/FSoE Inputs/FSOE/FSoE CRC 002
//     PlcTask Inputs/GVL_iXlinker.EtherCAT_Master_EKxxxx.Beckhoff_EKx9xx.Beckhoff_EKx9xxEK1122.A_0003_EK1960_0008_0019.Module_1_FSoE.FSoE_Inputs.FSOE/FSIN_Module_9_Module_Fault_1 <-> Module 1 (FSoE)/FSoE Inputs/FSOE/FSIN Module 9.Module Fault 1
//     PlcTask Inputs/GVL_iXlinker.EtherCAT_Master_EKxxxx.Beckhoff_EKx9xx.Beckhoff_EKx9xxEK1122.A_0003_EK1960_0008_0019.Module_1_FSoE.FSoE_Inputs.FSOE/FSIN_Module_9_Module_Fault_2 <-> Module 1 (FSoE)/FSoE Inputs/FSOE/FSIN Module 9.Module Fault 2
//     PlcTask Inputs/GVL_iXlinker.EtherCAT_Master_EKxxxx.Beckhoff_EKx9xx.Beckhoff_EKx9xxEK1122.A_0003_EK1960_0008_0019.Module_1_FSoE.FSoE_Inputs.FSOE/FSIN_Module_10_Module_Fault_1 <-> Module 1 (FSoE)/FSoE Inputs/FSOE/FSIN Module 10.Module Fault 1
//     PlcTask Inputs/GVL_iXlinker.EtherCAT_Master_EKxxxx.Beckhoff_EKx9xx.Beckhoff_EKx9xxEK1122.A_0003_EK1960_0008_0019.Module_1_FSoE.FSoE_Inputs.FSOE/FSIN_Module_10_Module_Fault_2 <-> Module 1 (FSoE)/FSoE Inputs/FSOE/FSIN Module 10.Module Fault 2
//     PlcTask Inputs/GVL_iXlinker.EtherCAT_Master_EKxxxx.Beckhoff_EKx9xx.Beckhoff_EKx9xxEK1122.A_0003_EK1960_0008_0019.Module_1_FSoE.FSoE_Inputs.FSOE/FSoE_Connection_ID <-> Module 1 (FSoE)/FSoE Inputs/FSOE/FSoE Connection ID
//     PlcTask Outputs/GVL_iXlinker.EtherCAT_Master_EKxxxx.Beckhoff_EKx9xx.Beckhoff_EKx9xxEK1122.A_0003_EK1960_0008_0019.Module_1_FSoE.FSoE_Outputs.FSOE/FSoE_Command <-> Module 1 (FSoE)/FSoE Outputs/FSOE/FSoE Command
//     PlcTask Outputs/GVL_iXlinker.EtherCAT_Master_EKxxxx.Beckhoff_EKx9xx.Beckhoff_EKx9xxEK1122.A_0003_EK1960_0008_0019.Module_1_FSoE.FSoE_Outputs.FSOE/FSOUT_Module_1_Channel_1_Output <-> Module 1 (FSoE)/FSoE Outputs/FSOE/FSOUT Module 1.Channel 1.Output
//     PlcTask Outputs/GVL_iXlinker.EtherCAT_Master_EKxxxx.Beckhoff_EKx9xx.Beckhoff_EKx9xxEK1122.A_0003_EK1960_0008_0019.Module_1_FSoE.FSoE_Outputs.FSOE/FSOUT_Module_1_Channel_2_Output <-> Module 1 (FSoE)/FSoE Outputs/FSOE/FSOUT Module 1.Channel 2.Output
//     PlcTask Outputs/GVL_iXlinker.EtherCAT_Master_EKxxxx.Beckhoff_EKx9xx.Beckhoff_EKx9xxEK1122.A_0003_EK1960_0008_0019.Module_1_FSoE.FSoE_Outputs.FSOE/FSOUT_Module_1_Channel_3_Output <-> Module 1 (FSoE)/FSoE Outputs/FSOE/FSOUT Module 1.Channel 3.Output
//     PlcTask Outputs/GVL_iXlinker.EtherCAT_Master_EKxxxx.Beckhoff_EKx9xx.Beckhoff_EKx9xxEK1122.A_0003_EK1960_0008_0019.Module_1_FSoE.FSoE_Outputs.FSOE/FSOUT_Module_1_Channel_4_Output <-> Module 1 (FSoE)/FSoE Outputs/FSOE/FSOUT Module 1.Channel 4.Output
//     PlcTask Outputs/GVL_iXlinker.EtherCAT_Master_EKxxxx.Beckhoff_EKx9xx.Beckhoff_EKx9xxEK1122.A_0003_EK1960_0008_0019.Module_1_FSoE.FSoE_Outputs.FSOE/FSOUT_Module_2_Channel_1_Output <-> Module 1 (FSoE)/FSoE Outputs/FSOE/FSOUT Module 2.Channel 1.Output
//     PlcTask Outputs/GVL_iXlinker.EtherCAT_Master_EKxxxx.Beckhoff_EKx9xx.Beckhoff_EKx9xxEK1122.A_0003_EK1960_0008_0019.Module_1_FSoE.FSoE_Outputs.FSOE/FSOUT_Module_2_Channel_2_Output <-> Module 1 (FSoE)/FSoE Outputs/FSOE/FSOUT Module 2.Channel 2.Output
//     PlcTask Outputs/GVL_iXlinker.EtherCAT_Master_EKxxxx.Beckhoff_EKx9xx.Beckhoff_EKx9xxEK1122.A_0003_EK1960_0008_0019.Module_1_FSoE.FSoE_Outputs.FSOE/FSOUT_Module_2_Channel_3_Output <-> Module 1 (FSoE)/FSoE Outputs/FSOE/FSOUT Module 2.Channel 3.Output
//     PlcTask Outputs/GVL_iXlinker.EtherCAT_Master_EKxxxx.Beckhoff_EKx9xx.Beckhoff_EKx9xxEK1122.A_0003_EK1960_0008_0019.Module_1_FSoE.FSoE_Outputs.FSOE/FSOUT_Module_2_Channel_4_Output <-> Module 1 (FSoE)/FSoE Outputs/FSOE/FSOUT Module 2.Channel 4.Output
//     PlcTask Outputs/GVL_iXlinker.EtherCAT_Master_EKxxxx.Beckhoff_EKx9xx.Beckhoff_EKx9xxEK1122.A_0003_EK1960_0008_0019.Module_1_FSoE.FSoE_Outputs.FSOE/FSOUT_Module_3_Channel_1_Output <-> Module 1 (FSoE)/FSoE Outputs/FSOE/FSOUT Module 3.Channel 1.Output
//     PlcTask Outputs/GVL_iXlinker.EtherCAT_Master_EKxxxx.Beckhoff_EKx9xx.Beckhoff_EKx9xxEK1122.A_0003_EK1960_0008_0019.Module_1_FSoE.FSoE_Outputs.FSOE/FSOUT_Module_3_Channel_2_Output <-> Module 1 (FSoE)/FSoE Outputs/FSOE/FSOUT Module 3.Channel 2.Output
//     PlcTask Outputs/GVL_iXlinker.EtherCAT_Master_EKxxxx.Beckhoff_EKx9xx.Beckhoff_EKx9xxEK1122.A_0003_EK1960_0008_0019.Module_1_FSoE.FSoE_Outputs.FSOE/FSOUT_Module_3_Channel_3_Output <-> Module 1 (FSoE)/FSoE Outputs/FSOE/FSOUT Module 3.Channel 3.Output
//     PlcTask Outputs/GVL_iXlinker.EtherCAT_Master_EKxxxx.Beckhoff_EKx9xx.Beckhoff_EKx9xxEK1122.A_0003_EK1960_0008_0019.Module_1_FSoE.FSoE_Outputs.FSOE/FSOUT_Module_3_Channel_4_Output <-> Module 1 (FSoE)/FSoE Outputs/FSOE/FSOUT Module 3.Channel 4.Output
//     PlcTask Outputs/GVL_iXlinker.EtherCAT_Master_EKxxxx.Beckhoff_EKx9xx.Beckhoff_EKx9xxEK1122.A_0003_EK1960_0008_0019.Module_1_FSoE.FSoE_Outputs.FSOE/FSOUT_Module_4_Channel_1_Output <-> Module 1 (FSoE)/FSoE Outputs/FSOE/FSOUT Module 4.Channel 1.Output
//     PlcTask Outputs/GVL_iXlinker.EtherCAT_Master_EKxxxx.Beckhoff_EKx9xx.Beckhoff_EKx9xxEK1122.A_0003_EK1960_0008_0019.Module_1_FSoE.FSoE_Outputs.FSOE/FSOUT_Module_4_Channel_2_Output <-> Module 1 (FSoE)/FSoE Outputs/FSOE/FSOUT Module 4.Channel 2.Output
//     PlcTask Outputs/GVL_iXlinker.EtherCAT_Master_EKxxxx.Beckhoff_EKx9xx.Beckhoff_EKx9xxEK1122.A_0003_EK1960_0008_0019.Module_1_FSoE.FSoE_Outputs.FSOE/FSOUT_Module_4_Channel_3_Output <-> Module 1 (FSoE)/FSoE Outputs/FSOE/FSOUT Module 4.Channel 3.Output
//     PlcTask Outputs/GVL_iXlinker.EtherCAT_Master_EKxxxx.Beckhoff_EKx9xx.Beckhoff_EKx9xxEK1122.A_0003_EK1960_0008_0019.Module_1_FSoE.FSoE_Outputs.FSOE/FSOUT_Module_4_Channel_4_Output <-> Module 1 (FSoE)/FSoE Outputs/FSOE/FSOUT Module 4.Channel 4.Output
//     PlcTask Outputs/GVL_iXlinker.EtherCAT_Master_EKxxxx.Beckhoff_EKx9xx.Beckhoff_EKx9xxEK1122.A_0003_EK1960_0008_0019.Module_1_FSoE.FSoE_Outputs.FSOE/FSOUT_Module_5_Channel_1_Output <-> Module 1 (FSoE)/FSoE Outputs/FSOE/FSOUT Module 5.Channel 1.Output
//     PlcTask Outputs/GVL_iXlinker.EtherCAT_Master_EKxxxx.Beckhoff_EKx9xx.Beckhoff_EKx9xxEK1122.A_0003_EK1960_0008_0019.Module_1_FSoE.FSoE_Outputs.FSOE/FSOUT_Module_5_Channel_2_Output <-> Module 1 (FSoE)/FSoE Outputs/FSOE/FSOUT Module 5.Channel 2.Output
//     PlcTask Outputs/GVL_iXlinker.EtherCAT_Master_EKxxxx.Beckhoff_EKx9xx.Beckhoff_EKx9xxEK1122.A_0003_EK1960_0008_0019.Module_1_FSoE.FSoE_Outputs.FSOE/FSOUT_Module_5_Channel_3_Output <-> Module 1 (FSoE)/FSoE Outputs/FSOE/FSOUT Module 5.Channel 3.Output
//     PlcTask Outputs/GVL_iXlinker.EtherCAT_Master_EKxxxx.Beckhoff_EKx9xx.Beckhoff_EKx9xxEK1122.A_0003_EK1960_0008_0019.Module_1_FSoE.FSoE_Outputs.FSOE/FSOUT_Module_5_Channel_4_Output <-> Module 1 (FSoE)/FSoE Outputs/FSOE/FSOUT Module 5.Channel 4.Output
//     PlcTask Outputs/GVL_iXlinker.EtherCAT_Master_EKxxxx.Beckhoff_EKx9xx.Beckhoff_EKx9xxEK1122.A_0003_EK1960_0008_0019.Module_1_FSoE.FSoE_Outputs.FSOE/FSOUT_Module_6_Channel_1_Output <-> Module 1 (FSoE)/FSoE Outputs/FSOE/FSOUT Module 6.Channel 1.Output
//     PlcTask Outputs/GVL_iXlinker.EtherCAT_Master_EKxxxx.Beckhoff_EKx9xx.Beckhoff_EKx9xxEK1122.A_0003_EK1960_0008_0019.Module_1_FSoE.FSoE_Outputs.FSOE/FSOUT_Module_6_Channel_2_Output <-> Module 1 (FSoE)/FSoE Outputs/FSOE/FSOUT Module 6.Channel 2.Output
//     PlcTask Outputs/GVL_iXlinker.EtherCAT_Master_EKxxxx.Beckhoff_EKx9xx.Beckhoff_EKx9xxEK1122.A_0003_EK1960_0008_0019.Module_1_FSoE.FSoE_Outputs.FSOE/FSOUT_Module_6_Channel_3_Output <-> Module 1 (FSoE)/FSoE Outputs/FSOE/FSOUT Module 6.Channel 3.Output
//     PlcTask Outputs/GVL_iXlinker.EtherCAT_Master_EKxxxx.Beckhoff_EKx9xx.Beckhoff_EKx9xxEK1122.A_0003_EK1960_0008_0019.Module_1_FSoE.FSoE_Outputs.FSOE/FSOUT_Module_6_Channel_4_Output <-> Module 1 (FSoE)/FSoE Outputs/FSOE/FSOUT Module 6.Channel 4.Output
//     PlcTask Outputs/GVL_iXlinker.EtherCAT_Master_EKxxxx.Beckhoff_EKx9xx.Beckhoff_EKx9xxEK1122.A_0003_EK1960_0008_0019.Module_1_FSoE.FSoE_Outputs.FSOE/FSOUT_Module_1_ErrAck <-> Module 1 (FSoE)/FSoE Outputs/FSOE/FSOUT Module 1.ErrAck
//     PlcTask Outputs/GVL_iXlinker.EtherCAT_Master_EKxxxx.Beckhoff_EKx9xx.Beckhoff_EKx9xxEK1122.A_0003_EK1960_0008_0019.Module_1_FSoE.FSoE_Outputs.FSOE/FSOUT_Module_2_ErrAck <-> Module 1 (FSoE)/FSoE Outputs/FSOE/FSOUT Module 2.ErrAck
//     PlcTask Outputs/GVL_iXlinker.EtherCAT_Master_EKxxxx.Beckhoff_EKx9xx.Beckhoff_EKx9xxEK1122.A_0003_EK1960_0008_0019.Module_1_FSoE.FSoE_Outputs.FSOE/FSOUT_Module_3_ErrAck <-> Module 1 (FSoE)/FSoE Outputs/FSOE/FSOUT Module 3.ErrAck
//     PlcTask Outputs/GVL_iXlinker.EtherCAT_Master_EKxxxx.Beckhoff_EKx9xx.Beckhoff_EKx9xxEK1122.A_0003_EK1960_0008_0019.Module_1_FSoE.FSoE_Outputs.FSOE/FSOUT_Module_4_ErrAck <-> Module 1 (FSoE)/FSoE Outputs/FSOE/FSOUT Module 4.ErrAck
//     PlcTask Outputs/GVL_iXlinker.EtherCAT_Master_EKxxxx.Beckhoff_EKx9xx.Beckhoff_EKx9xxEK1122.A_0003_EK1960_0008_0019.Module_1_FSoE.FSoE_Outputs.FSOE/FSOUT_Module_5_ErrAck <-> Module 1 (FSoE)/FSoE Outputs/FSOE/FSOUT Module 5.ErrAck
//     PlcTask Outputs/GVL_iXlinker.EtherCAT_Master_EKxxxx.Beckhoff_EKx9xx.Beckhoff_EKx9xxEK1122.A_0003_EK1960_0008_0019.Module_1_FSoE.FSoE_Outputs.FSOE/FSOUT_Module_6_ErrAck <-> Module 1 (FSoE)/FSoE Outputs/FSOE/FSOUT Module 6.ErrAck
//     PlcTask Outputs/GVL_iXlinker.EtherCAT_Master_EKxxxx.Beckhoff_EKx9xx.Beckhoff_EKx9xxEK1122.A_0003_EK1960_0008_0019.Module_1_FSoE.FSoE_Outputs.FSOE/FSoE_CRC_000 <-> Module 1 (FSoE)/FSoE Outputs/FSOE/FSoE CRC 000
//     PlcTask Outputs/GVL_iXlinker.EtherCAT_Master_EKxxxx.Beckhoff_EKx9xx.Beckhoff_EKx9xxEK1122.A_0003_EK1960_0008_0019.Module_1_FSoE.FSoE_Outputs.FSOE/FSoE_CRC_001 <-> Module 1 (FSoE)/FSoE Outputs/FSOE/FSoE CRC 001
//     PlcTask Outputs/GVL_iXlinker.EtherCAT_Master_EKxxxx.Beckhoff_EKx9xx.Beckhoff_EKx9xxEK1122.A_0003_EK1960_0008_0019.Module_1_FSoE.FSoE_Outputs.FSOE/FSoE_CRC_002 <-> Module 1 (FSoE)/FSoE Outputs/FSOE/FSoE CRC 002
//     PlcTask Outputs/GVL_iXlinker.EtherCAT_Master_EKxxxx.Beckhoff_EKx9xx.Beckhoff_EKx9xxEK1122.A_0003_EK1960_0008_0019.Module_1_FSoE.FSoE_Outputs.FSOE/FSIN_Module_1_ErrAck <-> Module 1 (FSoE)/FSoE Outputs/FSOE/FSIN Module 1.ErrAck
//     PlcTask Outputs/GVL_iXlinker.EtherCAT_Master_EKxxxx.Beckhoff_EKx9xx.Beckhoff_EKx9xxEK1122.A_0003_EK1960_0008_0019.Module_1_FSoE.FSoE_Outputs.FSOE/FSIN_Module_2_ErrAck <-> Module 1 (FSoE)/FSoE Outputs/FSOE/FSIN Module 2.ErrAck
//     PlcTask Outputs/GVL_iXlinker.EtherCAT_Master_EKxxxx.Beckhoff_EKx9xx.Beckhoff_EKx9xxEK1122.A_0003_EK1960_0008_0019.Module_1_FSoE.FSoE_Outputs.FSOE/FSIN_Module_3_ErrAck <-> Module 1 (FSoE)/FSoE Outputs/FSOE/FSIN Module 3.ErrAck
//     PlcTask Outputs/GVL_iXlinker.EtherCAT_Master_EKxxxx.Beckhoff_EKx9xx.Beckhoff_EKx9xxEK1122.A_0003_EK1960_0008_0019.Module_1_FSoE.FSoE_Outputs.FSOE/FSIN_Module_4_ErrAck <-> Module 1 (FSoE)/FSoE Outputs/FSOE/FSIN Module 4.ErrAck
//     PlcTask Outputs/GVL_iXlinker.EtherCAT_Master_EKxxxx.Beckhoff_EKx9xx.Beckhoff_EKx9xxEK1122.A_0003_EK1960_0008_0019.Module_1_FSoE.FSoE_Outputs.FSOE/FSIN_Module_5_ErrAck <-> Module 1 (FSoE)/FSoE Outputs/FSOE/FSIN Module 5.ErrAck
//     PlcTask Outputs/GVL_iXlinker.EtherCAT_Master_EKxxxx.Beckhoff_EKx9xx.Beckhoff_EKx9xxEK1122.A_0003_EK1960_0008_0019.Module_1_FSoE.FSoE_Outputs.FSOE/FSIN_Module_6_ErrAck <-> Module 1 (FSoE)/FSoE Outputs/FSOE/FSIN Module 6.ErrAck
//     PlcTask Outputs/GVL_iXlinker.EtherCAT_Master_EKxxxx.Beckhoff_EKx9xx.Beckhoff_EKx9xxEK1122.A_0003_EK1960_0008_0019.Module_1_FSoE.FSoE_Outputs.FSOE/FSIN_Module_7_ErrAck <-> Module 1 (FSoE)/FSoE Outputs/FSOE/FSIN Module 7.ErrAck
//     PlcTask Outputs/GVL_iXlinker.EtherCAT_Master_EKxxxx.Beckhoff_EKx9xx.Beckhoff_EKx9xxEK1122.A_0003_EK1960_0008_0019.Module_1_FSoE.FSoE_Outputs.FSOE/FSIN_Module_8_ErrAck <-> Module 1 (FSoE)/FSoE Outputs/FSOE/FSIN Module 8.ErrAck
//     PlcTask Outputs/GVL_iXlinker.EtherCAT_Master_EKxxxx.Beckhoff_EKx9xx.Beckhoff_EKx9xxEK1122.A_0003_EK1960_0008_0019.Module_1_FSoE.FSoE_Outputs.FSOE/FSIN_Module_9_ErrAck_1 <-> Module 1 (FSoE)/FSoE Outputs/FSOE/FSIN Module 9.ErrAck 1
//     PlcTask Outputs/GVL_iXlinker.EtherCAT_Master_EKxxxx.Beckhoff_EKx9xx.Beckhoff_EKx9xxEK1122.A_0003_EK1960_0008_0019.Module_1_FSoE.FSoE_Outputs.FSOE/FSIN_Module_9_ErrAck_2 <-> Module 1 (FSoE)/FSoE Outputs/FSOE/FSIN Module 9.ErrAck 2
//     PlcTask Outputs/GVL_iXlinker.EtherCAT_Master_EKxxxx.Beckhoff_EKx9xx.Beckhoff_EKx9xxEK1122.A_0003_EK1960_0008_0019.Module_1_FSoE.FSoE_Outputs.FSOE/FSIN_Module_10_ErrAck_1 <-> Module 1 (FSoE)/FSoE Outputs/FSOE/FSIN Module 10.ErrAck 1
//     PlcTask Outputs/GVL_iXlinker.EtherCAT_Master_EKxxxx.Beckhoff_EKx9xx.Beckhoff_EKx9xxEK1122.A_0003_EK1960_0008_0019.Module_1_FSoE.FSoE_Outputs.FSOE/FSIN_Module_10_ErrAck_2 <-> Module 1 (FSoE)/FSoE Outputs/FSOE/FSIN Module 10.ErrAck 2
//     PlcTask Outputs/GVL_iXlinker.EtherCAT_Master_EKxxxx.Beckhoff_EKx9xx.Beckhoff_EKx9xxEK1122.A_0003_EK1960_0008_0019.Module_1_FSoE.FSoE_Outputs.FSOE/FSoE_Connection_ID <-> Module 1 (FSoE)/FSoE Outputs/FSOE/FSoE Connection ID
//     PlcTask Outputs/GVL_iXlinker.EtherCAT_Master_EKxxxx.Beckhoff_EKx9xx.Beckhoff_EKx9xxEK1122.A_0003_EK1960_0008_0019.Module_2_FSOUT.Outputs.Module_1_Channel_1_Standard_Output_X5_1 <-> Module 2 (FSOUT)/Outputs/Module 1.Channel 1.Standard Output (X5.1)
//     PlcTask Outputs/GVL_iXlinker.EtherCAT_Master_EKxxxx.Beckhoff_EKx9xx.Beckhoff_EKx9xxEK1122.A_0003_EK1960_0008_0019.Module_2_FSOUT.Outputs.Module_1_Channel_2_Standard_Output_X5_2 <-> Module 2 (FSOUT)/Outputs/Module 1.Channel 2.Standard Output (X5.2)
//     PlcTask Outputs/GVL_iXlinker.EtherCAT_Master_EKxxxx.Beckhoff_EKx9xx.Beckhoff_EKx9xxEK1122.A_0003_EK1960_0008_0019.Module_2_FSOUT.Outputs.Module_1_Channel_3_Standard_Output_X5_3 <-> Module 2 (FSOUT)/Outputs/Module 1.Channel 3.Standard Output (X5.3)
//     PlcTask Outputs/GVL_iXlinker.EtherCAT_Master_EKxxxx.Beckhoff_EKx9xx.Beckhoff_EKx9xxEK1122.A_0003_EK1960_0008_0019.Module_2_FSOUT.Outputs.Module_1_Channel_4_Standard_Output_X5_4 <-> Module 2 (FSOUT)/Outputs/Module 1.Channel 4.Standard Output (X5.4)
//     PlcTask Outputs/GVL_iXlinker.EtherCAT_Master_EKxxxx.Beckhoff_EKx9xx.Beckhoff_EKx9xxEK1122.A_0003_EK1960_0008_0019.Module_2_FSOUT.Outputs.Module_2_Channel_1_Standard_Output_X5_5 <-> Module 2 (FSOUT)/Outputs/Module 2.Channel 1.Standard Output (X5.5)
